LIN {X 0,Y 472.884,Z 110.578,A -85,B 0,C 180,E1 22845.551,E2 22845.551} C_VEL
LIN {X 0,Y 472.896,Z 110.565,A -85,B 0,C 180,E1 22842.019,E2 22842.019} C_VEL
LIN {X 0,Y 472.934,Z 110.57,A -85,B 0,C 180,E1 22838.468,E2 22838.468} C_VEL
LIN {X 0,Y 472.917,Z 110.572,A -85,B 0,C 180,E1 22834.851,E2 22834.851} C_VEL
LIN {X 0,Y 472.886,Z 110.562,A -85,B 0,C 180,E1 22831.317,E2 22831.317} C_VEL
LIN {X 0,Y 472.877,Z 110.572,A -85,B 0,C 180,E1 22827.752,E2 22827.752} C_VEL
LIN {X 0,Y 472.902,Z 110.576,A -85,B 0,C 180,E1 22824.279,E2 22824.279} C_VEL
LIN {X 0,Y 472.936,Z 110.577,A -85,B 0,C 180,E1 22820.636,E2 22820.636} C_VEL
LIN {X 0,Y 472.912,Z 110.58,A -85,B 0,C 180,E1 22817.014,E2 22817.014} C_VEL
LIN {X 0,Y 472.879,Z 110.58,A -85,B 0,C 180,E1 22813.511,E2 22813.511} C_VEL
LIN {X 0,Y 472.876,Z 110.577,A -85,B 0,C 180,E1 22809.867,E2 22809.867} C_VEL
LIN {X 0,Y 472.932,Z 110.708,A -85,B 0,C 180,E1 22806.545,E2 22806.545} C_VEL
LIN {X 0,Y 480.969,Z 132.457,A -85,B 0,C 180,E1 22803.528,E2 22803.528} C_VEL
LIN {X 0,Y 484.768,Z 144.05,A -85,B 0,C 180,E1 22802.036,E2 22802.036} C_VEL
LIN {X 0,Y 482.911,Z 174.424,A -85,B 0,C 180,E1 22799.238,E2 22799.238} C_VEL
LIN {X 0,Y 483.355,Z 176.82,A -85,B 0,C 180,E1 22799.166,E2 22799.166} C_VEL
LIN {X 0,Y 483.697,Z 184.5,A -85,B 0,C 180,E1 22799.017,E2 22799.017} C_VEL
LIN {X 0,Y 481.966,Z 196.735,A -85,B 0,C 180,E1 22798.947,E2 22798.947} C_VEL
LIN {X 0,Y 480.031,Z 209.081,A -85,B 0,C 180,E1 22798.891,E2 22798.891} C_VEL
LIN {X 0,Y 479.862,Z 212.462,A -85,B 0,C 180,E1 22798.849,E2 22798.849} C_VEL
LIN {X 0,Y 477.924,Z 389.612,A -85,B 0,C 180,E1 22796.211,E2 22796.211} C_VEL
LIN {X 0,Y 477.296,Z 408.622,A -85,B 0,C 180,E1 22795.702,E2 22795.702} C_VEL
LIN {X 0,Y 476.379,Z 426.597,A -85,B 0,C 180,E1 22794.998,E2 22794.998} C_VEL
LIN {X 0,Y 475.201,Z 443.939,A -85,B 0,C 180,E1 22794.09,E2 22794.09} C_VEL
LIN {X 0,Y 473.813,Z 460.62,A -85,B 0,C 180,E1 22792.978,E2 22792.978} C_VEL
LIN {X 0,Y 472.296,Z 476.507,A -85,B 0,C 180,E1 22791.662,E2 22791.662} C_VEL
LIN {X 0,Y 470.707,Z 491.623,A -85,B 0,C 180,E1 22790.127,E2 22790.127} C_VEL
LIN {X 0,Y 469.264,Z 504.803,A -85,B 0,C 180,E1 22788.509,E2 22788.509} C_VEL
LIN {X 0,Y 467.857,Z 517.403,A -85,B 0,C 180,E1 22786.64,E2 22786.64} C_VEL
LIN {X 0,Y 466.665,Z 528.464,A -85,B 0,C 180,E1 22784.644,E2 22784.644} C_VEL
LIN {X 0,Y 465.712,Z 538.034,A -85,B 0,C 180,E1 22782.523,E2 22782.523} C_VEL
LIN {X 0,Y 465.004,Z 546.099,A -85,B 0,C 180,E1 22780.28,E2 22780.28} C_VEL
LIN {X 0,Y 464.565,Z 552.332,A -85,B 0,C 180,E1 22778.041,E2 22778.041} C_VEL
LIN {X 0,Y 464.288,Z 557.107,A -85,B 0,C 180,E1 22775.684,E2 22775.684} C_VEL
LIN {X 0,Y 464.151,Z 560.185,A -85,B 0,C 180,E1 22773.334,E2 22773.334} C_VEL
LIN {X 0,Y 464.105,Z 561.659,A -85,B 0,C 180,E1 22770.987,E2 22770.987} C_VEL
LIN {X 0,Y 464.108,Z 561.574,A -85,B 0,C 180,E1 22768.641,E2 22768.641} C_VEL
LIN {X 0,Y 464.165,Z 559.923,A -85,B 0,C 180,E1 22766.294,E2 22766.294} C_VEL
LIN {X 0,Y 464.318,Z 556.648,A -85,B 0,C 180,E1 22763.942,E2 22763.942} C_VEL
LIN {X 0,Y 464.611,Z 551.647,A -85,B 0,C 180,E1 22761.584,E2 22761.584} C_VEL
LIN {X 0,Y 465.118,Z 544.77,A -85,B 0,C 180,E1 22759.22,E2 22759.22} C_VEL
LIN {X 0,Y 465.876,Z 536.323,A -85,B 0,C 180,E1 22756.976,E2 22756.976} C_VEL
LIN {X 0,Y 466.882,Z 526.333,A -85,B 0,C 180,E1 22754.854,E2 22754.854} C_VEL
LIN {X 0,Y 468.047,Z 515.598,A -85,B 0,C 180,E1 22752.982,E2 22752.982} C_VEL
LIN {X 0,Y 469.446,Z 503.079,A -85,B 0,C 180,E1 22751.175,E2 22751.175} C_VEL
LIN {X 0,Y 470.928,Z 489.575,A -85,B 0,C 180,E1 22749.557,E2 22749.557} C_VEL
LIN {X 0,Y 472.43,Z 475.214,A -85,B 0,C 180,E1 22748.13,E2 22748.13} C_VEL
LIN {X 0,Y 473.935,Z 459.24,A -85,B 0,C 180,E1 22746.829,E2 22746.829} C_VEL
LIN {X 0,Y 475.26,Z 443.306,A -85,B 0,C 180,E1 22745.779,E2 22745.779} C_VEL
LIN {X 0,Y 476.469,Z 425.323,A -85,B 0,C 180,E1 22744.852,E2 22744.852} C_VEL
LIN {X 0,Y 477.378,Z 406.697,A -85,B 0,C 180,E1 22744.143,E2 22744.143} C_VEL
LIN {X 0,Y 477.973,Z 387.762,A -85,B 0,C 180,E1 22743.661,E2 22743.661} C_VEL
LIN {X 0,Y 479.954,Z 196.45,A -85,B 0,C 180,E1 22740.803,E2 22740.803} C_VEL
LIN {X 0,Y 475.821,Z 173.604,A -85,B 0,C 180,E1 22740.096,E2 22740.096} C_VEL
LIN {X 0,Y 477.63,Z 146.449,A -85,B 0,C 180,E1 22737.526,E2 22737.526} C_VEL
LIN {X 0,Y 470.909,Z 127.236,A -85,B 0,C 180,E1 22734.937,E2 22734.937} C_VEL
LIN {X 0,Y 464.971,Z 111.558,A -85,B 0,C 180,E1 22732.631,E2 22732.631} C_VEL
LIN {X 0,Y 465.011,Z 111.552,A -85,B 0,C 180,E1 22729.181,E2 22729.181} C_VEL
LIN {X 0,Y 465.016,Z 111.564,A -85,B 0,C 180,E1 22725.496,E2 22725.496} C_VEL
LIN {X 0,Y 465.012,Z 111.562,A -85,B 0,C 180,E1 22721.744,E2 22721.744} C_VEL
LIN {X 0,Y 465.009,Z 111.563,A -85,B 0,C 180,E1 22718.096,E2 22718.096} C_VEL
LIN {X 0,Y 465.023,Z 111.688,A -85,B 0,C 180,E1 22715.488,E2 22715.488} C_VEL
LIN {X 0,Y 474.191,Z 138.149,A -85,B 0,C 180,E1 22712.496,E2 22712.496} C_VEL
LIN {X 0,Y 475.436,Z 142.809,A -85,B 0,C 180,E1 22712.003,E2 22712.003} C_VEL
LIN {X 0,Y 474.177,Z 181.693,A -85,B 0,C 180,E1 22708.738,E2 22708.738} C_VEL
LIN {X 0,Y 476.41,Z 196.928,A -85,B 0,C 180,E1 22708.313,E2 22708.313} C_VEL
LIN {X 0,Y 472.786,Z 392,A -85,B 0,C 180,E1 22704.905,E2 22704.905} C_VEL
LIN {X 0,Y 472.247,Z 411.513,A -85,B 0,C 180,E1 22704.331,E2 22704.331} C_VEL
LIN {X 0,Y 471.525,Z 429.876,A -85,B 0,C 180,E1 22703.56,E2 22703.56} C_VEL
LIN {X 0,Y 470.673,Z 447.161,A -85,B 0,C 180,E1 22702.613,E2 22702.613} C_VEL
LIN {X 0,Y 469.738,Z 463.701,A -85,B 0,C 180,E1 22701.476,E2 22701.476} C_VEL
LIN {X 0,Y 468.755,Z 479.425,A -85,B 0,C 180,E1 22700.15,E2 22700.15} C_VEL
LIN {X 0,Y 467.767,Z 494.215,A -85,B 0,C 180,E1 22698.637,E2 22698.637} C_VEL
LIN {X 0,Y 466.826,Z 507.992,A -85,B 0,C 180,E1 22696.935,E2 22696.935} C_VEL
LIN {X 0,Y 465.986,Z 520.624,A -85,B 0,C 180,E1 22695.048,E2 22695.048} C_VEL
LIN {X 0,Y 465.347,Z 531.015,A -85,B 0,C 180,E1 22693.165,E2 22693.165} C_VEL
LIN {X 0,Y 464.851,Z 540.065,A -85,B 0,C 180,E1 22691.162,E2 22691.162} C_VEL
LIN {X 0,Y 464.502,Z 547.713,A -85,B 0,C 180,E1 22689.041,E2 22689.041} C_VEL
LIN {X 0,Y 464.287,Z 553.881,A -85,B 0,C 180,E1 22686.803,E2 22686.803} C_VEL
LIN {X 0,Y 464.162,Z 558.237,A -85,B 0,C 180,E1 22684.572,E2 22684.572} C_VEL
LIN {X 0,Y 464.122,Z 560.897,A -85,B 0,C 180,E1 22682.346,E2 22682.346} C_VEL
LIN {X 0,Y 464.117,Z 561.965,A -85,B 0,C 180,E1 22680,E2 22680} C_VEL
LIN {X 0,Y 464.137,Z 561.22,A -85,B 0,C 180,E1 22677.654,E2 22677.654} C_VEL
LIN {X 0,Y 464.202,Z 558.846,A -85,B 0,C 180,E1 22675.429,E2 22675.429} C_VEL
LIN {X 0,Y 464.341,Z 554.769,A -85,B 0,C 180,E1 22673.199,E2 22673.199} C_VEL
LIN {X 0,Y 464.581,Z 548.874,A -85,B 0,C 180,E1 22670.961,E2 22670.961} C_VEL
LIN {X 0,Y 464.95,Z 541.471,A -85,B 0,C 180,E1 22668.841,E2 22668.841} C_VEL
LIN {X 0,Y 465.464,Z 532.625,A -85,B 0,C 180,E1 22666.839,E2 22666.839} C_VEL
LIN {X 0,Y 466.153,Z 521.688,A -85,B 0,C 180,E1 22664.844,E2 22664.844} C_VEL
LIN {X 0,Y 466.941,Z 509.853,A -85,B 0,C 180,E1 22663.069,E2 22663.069} C_VEL
LIN {X 0,Y 467.832,Z 496.357,A -85,B 0,C 180,E1 22661.398,E2 22661.398} C_VEL
LIN {X 0,Y 468.744,Z 481.822,A -85,B 0,C 180,E1 22659.915,E2 22659.915} C_VEL
LIN {X 0,Y 469.664,Z 466.017,A -85,B 0,C 180,E1 22658.586,E2 22658.586} C_VEL
LIN {X 0,Y 470.528,Z 449.162,A -85,B 0,C 180,E1 22657.441,E2 22657.441} C_VEL
LIN {X 0,Y 471.258,Z 431.359,A -85,B 0,C 180,E1 22656.492,E2 22656.492} C_VEL
LIN {X 0,Y 471.838,Z 412.338,A -85,B 0,C 180,E1 22655.73,E2 22655.73} C_VEL
LIN {X 0,Y 472.248,Z 392.418,A -85,B 0,C 180,E1 22655.181,E2 22655.181} C_VEL
LIN {X 0,Y 474.476,Z 285.661,A -85,B 0,C 180,E1 22653.199,E2 22653.199} C_VEL
LIN {X 0,Y 477.349,Z 195.104,A -85,B 0,C 180,E1 22651.339,E2 22651.339} C_VEL
LIN {X 0,Y 476.497,Z 189.323,A -85,B 0,C 180,E1 22651.106,E2 22651.106} C_VEL
LIN {X 0,Y 477.357,Z 150.37,A -85,B 0,C 180,E1 22648,E2 22648} C_VEL
LIN {X 0,Y 477.285,Z 141.627,A -85,B 0,C 180,E1 22647.284,E2 22647.284} C_VEL
LIN {X 0,Y 473.092,Z 129.321,A -85,B 0,C 180,E1 22645.835,E2 22645.835} C_VEL
LIN {X 0,Y 468.871,Z 119.813,A -85,B 0,C 180,E1 22644.547,E2 22644.547} C_VEL
LIN {X 0,Y 466.651,Z 115.532,A -85,B 0,C 180,E1 22643.898,E2 22643.898} C_VEL
LIN {X 0,Y 465.172,Z 112.443,A -85,B 0,C 180,E1 22643.429,E2 22643.429} C_VEL
LIN {X 0,Y 465.004,Z 111.566,A -85,B 0,C 180,E1 22643.291,E2 22643.291} C_VEL
LIN {X 0,Y 465.017,Z 111.564,A -85,B 0,C 180,E1 22639.567,E2 22639.567} C_VEL
LIN {X 0,Y 464.995,Z 111.566,A -85,B 0,C 180,E1 22635.839,E2 22635.839} C_VEL
LIN {X 0,Y 464.957,Z 111.57,A -85,B 0,C 180,E1 22632.29,E2 22632.29} C_VEL
LIN {X 0,Y 464.98,Z 111.74,A -85,B 0,C 180,E1 22631.259,E2 22631.259} C_VEL
LIN {X 0,Y 466.342,Z 115.196,A -85,B 0,C 180,E1 22630.813,E2 22630.813} C_VEL
LIN {X 0,Y 474.889,Z 135.664,A -85,B 0,C 180,E1 22628.244,E2 22628.244} C_VEL
LIN {X 0,Y 480.318,Z 150.221,A -85,B 0,C 180,E1 22626.579,E2 22626.579} C_VEL
LIN {X 0,Y 479.458,Z 164.644,A -85,B 0,C 180,E1 22625.503,E2 22625.503} C_VEL
LIN {X 0,Y 482.328,Z 186.5,A -85,B 0,C 180,E1 22624.889,E2 22624.889} C_VEL
LIN {X 0,Y 477.886,Z 419.576,A -85,B 0,C 180,E1 22620.981,E2 22620.981} C_VEL
LIN {X 0,Y 477.06,Z 440.311,A -85,B 0,C 180,E1 22620.457,E2 22620.457} C_VEL
LIN {X 0,Y 475.912,Z 461.474,A -85,B 0,C 180,E1 22619.697,E2 22619.697} C_VEL
LIN {X 0,Y 474.61,Z 482.255,A -85,B 0,C 180,E1 22618.707,E2 22618.707} C_VEL
LIN {X 0,Y 473.221,Z 501.389,A -85,B 0,C 180,E1 22617.564,E2 22617.564} C_VEL
LIN {X 0,Y 471.864,Z 519.025,A -85,B 0,C 180,E1 22616.287,E2 22616.287} C_VEL
LIN {X 0,Y 470.379,Z 537.148,A -85,B 0,C 180,E1 22614.713,E2 22614.713} C_VEL
LIN {X 0,Y 468.909,Z 554.52,A -85,B 0,C 180,E1 22612.905,E2 22612.905} C_VEL
LIN {X 0,Y 467.617,Z 569.978,A -85,B 0,C 180,E1 22610.987,E2 22610.987} C_VEL
LIN {X 0,Y 466.549,Z 583.421,A -85,B 0,C 180,E1 22609.012,E2 22609.012} C_VEL
LIN {X 0,Y 465.633,Z 595.835,A -85,B 0,C 180,E1 22606.852,E2 22606.852} C_VEL
LIN {X 0,Y 464.941,Z 606.773,A -85,B 0,C 180,E1 22604.573,E2 22604.573} C_VEL
LIN {X 0,Y 464.464,Z 615.766,A -85,B 0,C 180,E1 22602.306,E2 22602.306} C_VEL
LIN {X 0,Y 464.166,Z 623.312,A -85,B 0,C 180,E1 22599.924,E2 22599.924} C_VEL
LIN {X 0,Y 464,Z 629.057,A -85,B 0,C 180,E1 22597.554,E2 22597.554} C_VEL
LIN {X 0,Y 463.931,Z 633.365,A -85,B 0,C 180,E1 22595.07,E2 22595.07} C_VEL
LIN {X 0,Y 463.909,Z 635.899,A -85,B 0,C 180,E1 22592.719,E2 22592.719} C_VEL
LIN {X 0,Y 463.906,Z 636.873,A -85,B 0,C 180,E1 22590.248,E2 22590.248} C_VEL
LIN {X 0,Y 463.907,Z 636.257,A -85,B 0,C 180,E1 22587.901,E2 22587.901} C_VEL
LIN {X 0,Y 463.918,Z 634.033,A -85,B 0,C 180,E1 22585.427,E2 22585.427} C_VEL
LIN {X 0,Y 463.987,Z 630.124,A -85,B 0,C 180,E1 22582.945,E2 22582.945} C_VEL
LIN {X 0,Y 464.139,Z 624.343,A -85,B 0,C 180,E1 22580.453,E2 22580.453} C_VEL
LIN {X 0,Y 464.41,Z 617.058,A -85,B 0,C 180,E1 22578.073,E2 22578.073} C_VEL
LIN {X 0,Y 464.876,Z 607.875,A -85,B 0,C 180,E1 22575.681,E2 22575.681} C_VEL
LIN {X 0,Y 465.546,Z 597.191,A -85,B 0,C 180,E1 22573.403,E2 22573.403} C_VEL
LIN {X 0,Y 466.43,Z 585.055,A -85,B 0,C 180,E1 22571.245,E2 22571.245} C_VEL
LIN {X 0,Y 467.536,Z 571.073,A -85,B 0,C 180,E1 22569.156,E2 22569.156} C_VEL
LIN {X 0,Y 468.863,Z 555.12,A -85,B 0,C 180,E1 22567.164,E2 22567.164} C_VEL
LIN {X 0,Y 470.301,Z 538.046,A -85,B 0,C 180,E1 22565.375,E2 22565.375} C_VEL
LIN {X 0,Y 471.763,Z 520.178,A -85,B 0,C 180,E1 22563.807,E2 22563.807} C_VEL
LIN {X 0,Y 473.146,Z 502.356,A -85,B 0,C 180,E1 22562.502,E2 22562.502} C_VEL
LIN {X 0,Y 474.555,Z 483.031,A -85,B 0,C 180,E1 22561.335,E2 22561.335} C_VEL
LIN {X 0,Y 475.816,Z 463.201,A -85,B 0,C 180,E1 22560.375,E2 22560.375} C_VEL
LIN {X 0,Y 476.949,Z 442.8,A -85,B 0,C 180,E1 22559.617,E2 22559.617} C_VEL
LIN {X 0,Y 477.827,Z 421.76,A -85,B 0,C 180,E1 22559.06,E2 22559.06} C_VEL
LIN {X 0,Y 482.199,Z 192.981,A -85,B 0,C 180,E1 22555.217,E2 22555.217} C_VEL
LIN {X 0,Y 482.153,Z 183.797,A -85,B 0,C 180,E1 22555.048,E2 22555.048} C_VEL
LIN {X 0,Y 479.375,Z 163.766,A -85,B 0,C 180,E1 22554.465,E2 22554.465} C_VEL
LIN {X 0,Y 480.247,Z 149.701,A -85,B 0,C 180,E1 22553.379,E2 22553.379} C_VEL
LIN {X 0,Y 472.083,Z 128.682,A -85,B 0,C 180,E1 22550.917,E2 22550.917} C_VEL
LIN {X 0,Y 465.849,Z 114.357,A -85,B 0,C 180,E1 22549.069,E2 22549.069} C_VEL
LIN {X 0,Y 464.971,Z 111.558,A -85,B 0,C 180,E1 22548.689,E2 22548.689} C_VEL
LIN {X 0,Y 464.959,Z 111.567,A -85,B 0,C 180,E1 22545.145,E2 22545.145} C_VEL
LIN {X 0,Y 464.967,Z 111.565,A -85,B 0,C 180,E1 22541.477,E2 22541.477} C_VEL
LIN {X 0,Y 464.989,Z 111.522,A -85,B 0,C 180,E1 22537.895,E2 22537.895} C_VEL
LIN {X 0,Y 465.005,Z 111.562,A -85,B 0,C 180,E1 22534.288,E2 22534.288} C_VEL
LIN {X 0,Y 464.98,Z 111.565,A -85,B 0,C 180,E1 22530.639,E2 22530.639} C_VEL
LIN {X 0,Y 464.956,Z 111.564,A -85,B 0,C 180,E1 22527.094,E2 22527.094} C_VEL
LIN {X 0,Y 464.955,Z 111.557,A -85,B 0,C 180,E1 22523.442,E2 22523.442} C_VEL
LIN {X 0,Y 464.986,Z 111.555,A -85,B 0,C 180,E1 22519.992,E2 22519.992} C_VEL
LIN {X 0,Y 465.005,Z 111.562,A -85,B 0,C 180,E1 22516.36,E2 22516.36} C_VEL
LIN {X 0,Y 464.97,Z 111.547,A -85,B 0,C 180,E1 22512.796,E2 22512.796} C_VEL
LIN {X 0,Y 464.951,Z 111.564,A -85,B 0,C 180,E1 22509.234,E2 22509.234} C_VEL
LIN {X 0,Y 464.95,Z 111.563,A -85,B 0,C 180,E1 22505.553,E2 22505.553} C_VEL
LIN {X 0,Y 464.967,Z 111.552,A -85,B 0,C 180,E1 22501.971,E2 22501.971} C_VEL
LIN {X 0,Y 465.001,Z 111.562,A -85,B 0,C 180,E1 22498.398,E2 22498.398} C_VEL
LIN {X 0,Y 464.985,Z 111.547,A -85,B 0,C 180,E1 22494.694,E2 22494.694} C_VEL
LIN {X 0,Y 464.952,Z 111.566,A -85,B 0,C 180,E1 22491.217,E2 22491.217} C_VEL
LIN {X 0,Y 464.946,Z 111.557,A -85,B 0,C 180,E1 22487.581,E2 22487.581} C_VEL
LIN {X 0,Y 464.956,Z 111.56,A -85,B 0,C 180,E1 22483.993,E2 22483.993} C_VEL
LIN {X 0,Y 464.988,Z 111.563,A -85,B 0,C 180,E1 22480.4,E2 22480.4} C_VEL
LIN {X 0,Y 464.981,Z 111.549,A -85,B 0,C 180,E1 22476.827,E2 22476.827} C_VEL
LIN {X 0,Y 464.949,Z 111.565,A -85,B 0,C 180,E1 22473.291,E2 22473.291} C_VEL
LIN {X 0,Y 464.941,Z 111.566,A -85,B 0,C 180,E1 22469.787,E2 22469.787} C_VEL
LIN {X 0,Y 464.966,Z 111.558,A -85,B 0,C 180,E1 22466.303,E2 22466.303} C_VEL
LIN {X 0,Y 464.989,Z 111.555,A -85,B 0,C 180,E1 22462.671,E2 22462.671} C_VEL
LIN {X 0,Y 464.957,Z 111.561,A -85,B 0,C 180,E1 22459.176,E2 22459.176} C_VEL
LIN {X 0,Y 464.937,Z 111.56,A -85,B 0,C 180,E1 22455.659,E2 22455.659} C_VEL
LIN {X 0,Y 464.94,Z 111.571,A -85,B 0,C 180,E1 22451.92,E2 22451.92} C_VEL
LIN {X 0,Y 464.964,Z 111.566,A -85,B 0,C 180,E1 22448.422,E2 22448.422} C_VEL
LIN {X 0,Y 464.964,Z 111.582,A -85,B 0,C 180,E1 22447.234,E2 22447.234} C_VEL
LIN {X 0,Y 473.344,Z 133.939,A -85,B 0,C 180,E1 22444.039,E2 22444.039} C_VEL
LIN {X 0,Y 477.642,Z 146.882,A -85,B 0,C 180,E1 22442.332,E2 22442.332} C_VEL
LIN {X 0,Y 475.862,Z 174.32,A -85,B 0,C 180,E1 22439.775,E2 22439.775} C_VEL
LIN {X 0,Y 480.041,Z 198.192,A -85,B 0,C 180,E1 22439.066,E2 22439.066} C_VEL
LIN {X 0,Y 479.862,Z 212.462,A -85,B 0,C 180,E1 22438.849,E2 22438.849} C_VEL
LIN {X 0,Y 478.922,Z 220.158,A -85,B 0,C 180,E1 22438.796,E2 22438.796} C_VEL
LIN {X 0,Y 473.357,Z 240.654,A -85,B 0,C 180,E1 22438.882,E2 22438.882} C_VEL
LIN {X 0,Y 472.632,Z 247.261,A -85,B 0,C 180,E1 22438.83,E2 22438.83} C_VEL
LIN {X 0,Y 470.941,Z 389.942,A -85,B 0,C 180,E1 22436.681,E2 22436.681} C_VEL
LIN {X 0,Y 470.272,Z 408.97,A -85,B 0,C 180,E1 22436.166,E2 22436.166} C_VEL
LIN {X 0,Y 469.353,Z 426.237,A -85,B 0,C 180,E1 22435.487,E2 22435.487} C_VEL
LIN {X 0,Y 468.072,Z 444.088,A -85,B 0,C 180,E1 22434.548,E2 22434.548} C_VEL
LIN {X 0,Y 466.596,Z 460.843,A -85,B 0,C 180,E1 22433.421,E2 22433.421} C_VEL
LIN {X 0,Y 464.942,Z 477.199,A -85,B 0,C 180,E1 22432.048,E2 22432.048} C_VEL
LIN {X 0,Y 463.255,Z 492.276,A -85,B 0,C 180,E1 22430.492,E2 22430.492} C_VEL
LIN {X 0,Y 461.691,Z 505.63,A -85,B 0,C 180,E1 22428.824,E2 22428.824} C_VEL
LIN {X 0,Y 460.19,Z 518.191,A -85,B 0,C 180,E1 22426.925,E2 22426.925} C_VEL
LIN {X 0,Y 458.914,Z 529.22,A -85,B 0,C 180,E1 22424.897,E2 22424.897} C_VEL
LIN {X 0,Y 457.889,Z 538.763,A -85,B 0,C 180,E1 22422.74,E2 22422.74} C_VEL
LIN {X 0,Y 457.122,Z 546.805,A -85,B 0,C 180,E1 22420.459,E2 22420.459} C_VEL
LIN {X 0,Y 456.64,Z 553.016,A -85,B 0,C 180,E1 22418.181,E2 22418.181} C_VEL
LIN {X 0,Y 456.336,Z 557.773,A -85,B 0,C 180,E1 22415.784,E2 22415.784} C_VEL
LIN {X 0,Y 456.183,Z 560.838,A -85,B 0,C 180,E1 22413.392,E2 22413.392} C_VEL
LIN {X 0,Y 456.132,Z 562.305,A -85,B 0,C 180,E1 22411.004,E2 22411.004} C_VEL
LIN {X 0,Y 456.135,Z 562.22,A -85,B 0,C 180,E1 22408.618,E2 22408.618} C_VEL
LIN {X 0,Y 456.2,Z 560.578,A -85,B 0,C 180,E1 22406.229,E2 22406.229} C_VEL
LIN {X 0,Y 456.369,Z 557.318,A -85,B 0,C 180,E1 22403.836,E2 22403.836} C_VEL
LIN {X 0,Y 456.692,Z 552.337,A -85,B 0,C 180,E1 22401.437,E2 22401.437} C_VEL
LIN {X 0,Y 457.247,Z 545.482,A -85,B 0,C 180,E1 22399.032,E2 22399.032} C_VEL
LIN {X 0,Y 458.068,Z 537.062,A -85,B 0,C 180,E1 22396.75,E2 22396.75} C_VEL
LIN {X 0,Y 459.081,Z 527.764,A -85,B 0,C 180,E1 22394.719,E2 22394.719} C_VEL
LIN {X 0,Y 460.398,Z 516.398,A -85,B 0,C 180,E1 22392.69,E2 22392.69} C_VEL
LIN {X 0,Y 461.89,Z 503.92,A -85,B 0,C 180,E1 22390.855,E2 22390.855} C_VEL
LIN {X 0,Y 463.467,Z 490.469,A -85,B 0,C 180,E1 22389.213,E2 22389.213} C_VEL
LIN {X 0,Y 465.132,Z 475.466,A -85,B 0,C 180,E1 22387.702,E2 22387.702} C_VEL
LIN {X 0,Y 466.73,Z 459.427,A -85,B 0,C 180,E1 22386.383,E2 22386.383} C_VEL
LIN {X 0,Y 468.135,Z 443.413,A -85,B 0,C 180,E1 22385.319,E2 22385.319} C_VEL
LIN {X 0,Y 469.417,Z 425.305,A -85,B 0,C 180,E1 22384.38,E2 22384.38} C_VEL
LIN {X 0,Y 470.363,Z 407.017,A -85,B 0,C 180,E1 22383.678,E2 22383.678} C_VEL
LIN {X 0,Y 470.994,Z 388.14,A -85,B 0,C 180,E1 22383.191,E2 22383.191} C_VEL
LIN {X 0,Y 473.154,Z 197.742,A -85,B 0,C 180,E1 22380.307,E2 22380.307} C_VEL
LIN {X 0,Y 468.812,Z 173.404,A -85,B 0,C 180,E1 22379.531,E2 22379.531} C_VEL
LIN {X 0,Y 470.557,Z 149.679,A -85,B 0,C 180,E1 22377.263,E2 22377.263} C_VEL
LIN {X 0,Y 463.949,Z 130.687,A -85,B 0,C 180,E1 22374.658,E2 22374.658} C_VEL
LIN {X 0,Y 458.059,Z 115.586,A -85,B 0,C 180,E1 22372.407,E2 22372.407} C_VEL
LIN {X 0,Y 457.042,Z 112.527,A -85,B 0,C 180,E1 22371.907,E2 22371.907} C_VEL
LIN {X 0,Y 457.05,Z 112.558,A -85,B 0,C 180,E1 22368.244,E2 22368.244} C_VEL
LIN {X 0,Y 457.054,Z 112.552,A -85,B 0,C 180,E1 22364.506,E2 22364.506} C_VEL
LIN {X 0,Y 457.063,Z 112.55,A -85,B 0,C 180,E1 22360.808,E2 22360.808} C_VEL
LIN {X 0,Y 457.072,Z 112.549,A -85,B 0,C 180,E1 22357.14,E2 22357.14} C_VEL
LIN {X 0,Y 457.076,Z 112.659,A -85,B 0,C 180,E1 22356.012,E2 22356.012} C_VEL
LIN {X 0,Y 466.199,Z 138.753,A -85,B 0,C 180,E1 22353.008,E2 22353.008} C_VEL
LIN {X 0,Y 468.16,Z 145.565,A -85,B 0,C 180,E1 22352.272,E2 22352.272} C_VEL
LIN {X 0,Y 466.936,Z 182.274,A -85,B 0,C 180,E1 22349.18,E2 22349.18} C_VEL
LIN {X 0,Y 469.217,Z 197.998,A -85,B 0,C 180,E1 22348.726,E2 22348.726} C_VEL
LIN {X 0,Y 465.316,Z 392.645,A -85,B 0,C 180,E1 22345.248,E2 22345.248} C_VEL
LIN {X 0,Y 464.745,Z 412.117,A -85,B 0,C 180,E1 22344.663,E2 22344.663} C_VEL
LIN {X 0,Y 463.956,Z 430.969,A -85,B 0,C 180,E1 22343.854,E2 22343.854} C_VEL
LIN {X 0,Y 463.044,Z 448.433,A -85,B 0,C 180,E1 22342.873,E2 22342.873} C_VEL
LIN {X 0,Y 462.02,Z 465.459,A -85,B 0,C 180,E1 22341.669,E2 22341.669} C_VEL
LIN {X 0,Y 460.933,Z 481.828,A -85,B 0,C 180,E1 22340.242,E2 22340.242} C_VEL
LIN {X 0,Y 459.909,Z 496.366,A -85,B 0,C 180,E1 22338.704,E2 22338.704} C_VEL
LIN {X 0,Y 458.94,Z 509.938,A -85,B 0,C 180,E1 22336.974,E2 22336.974} C_VEL
LIN {X 0,Y 458.123,Z 521.619,A -85,B 0,C 180,E1 22335.183,E2 22335.183} C_VEL
LIN {X 0,Y 457.449,Z 531.987,A -85,B 0,C 180,E1 22333.268,E2 22333.268} C_VEL
LIN {X 0,Y 456.924,Z 541.002,A -85,B 0,C 180,E1 22331.231,E2 22331.231} C_VEL
LIN {X 0,Y 456.553,Z 548.611,A -85,B 0,C 180,E1 22329.073,E2 22329.073} C_VEL
LIN {X 0,Y 456.324,Z 554.737,A -85,B 0,C 180,E1 22326.795,E2 22326.795} C_VEL
LIN {X 0,Y 456.193,Z 559.047,A -85,B 0,C 180,E1 22324.526,E2 22324.526} C_VEL
LIN {X 0,Y 456.147,Z 561.743,A -85,B 0,C 180,E1 22322.136,E2 22322.136} C_VEL
LIN {X 0,Y 456.147,Z 562.631,A -85,B 0,C 180,E1 22319.875,E2 22319.875} C_VEL
LIN {X 0,Y 456.169,Z 561.903,A -85,B 0,C 180,E1 22317.613,E2 22317.613} C_VEL
LIN {X 0,Y 456.245,Z 559.537,A -85,B 0,C 180,E1 22315.349,E2 22315.349} C_VEL
LIN {X 0,Y 456.401,Z 555.462,A -85,B 0,C 180,E1 22313.08,E2 22313.08} C_VEL
LIN {X 0,Y 456.652,Z 549.935,A -85,B 0,C 180,E1 22310.928,E2 22310.928} C_VEL
LIN {X 0,Y 457.047,Z 542.607,A -85,B 0,C 180,E1 22308.773,E2 22308.773} C_VEL
LIN {X 0,Y 457.6,Z 533.846,A -85,B 0,C 180,E1 22306.737,E2 22306.737} C_VEL
LIN {X 0,Y 458.294,Z 523.711,A -85,B 0,C 180,E1 22304.823,E2 22304.823} C_VEL
LIN {X 0,Y 459.109,Z 512.192,A -85,B 0,C 180,E1 22303.033,E2 22303.033} C_VEL
LIN {X 0,Y 460.06,Z 498.707,A -85,B 0,C 180,E1 22301.303,E2 22301.303} C_VEL
LIN {X 0,Y 461.053,Z 484.195,A -85,B 0,C 180,E1 22299.764,E2 22299.764} C_VEL
LIN {X 0,Y 462.02,Z 468.677,A -85,B 0,C 180,E1 22298.414,E2 22298.414} C_VEL
LIN {X 0,Y 462.98,Z 451.328,A -85,B 0,C 180,E1 22297.192,E2 22297.192} C_VEL
LIN {X 0,Y 463.8,Z 433.347,A -85,B 0,C 180,E1 22296.192,E2 22296.192} C_VEL
LIN {X 0,Y 464.438,Z 414.471,A -85,B 0,C 180,E1 22295.407,E2 22295.407} C_VEL
LIN {X 0,Y 464.877,Z 395.153,A -85,B 0,C 180,E1 22294.846,E2 22294.846} C_VEL
LIN {X 0,Y 467.441,Z 286.91,A -85,B 0,C 180,E1 22292.75,E2 22292.75} C_VEL
LIN {X 0,Y 470.714,Z 196.563,A -85,B 0,C 180,E1 22290.821,E2 22290.821} C_VEL
LIN {X 0,Y 469.842,Z 190.427,A -85,B 0,C 180,E1 22290.555,E2 22290.555} C_VEL
LIN {X 0,Y 470.904,Z 150.854,A -85,B 0,C 180,E1 22287.363,E2 22287.363} C_VEL
LIN {X 0,Y 470.942,Z 145.552,A -85,B 0,C 180,E1 22286.932,E2 22286.932} C_VEL
LIN {X 0,Y 467.085,Z 133.878,A -85,B 0,C 180,E1 22285.503,E2 22285.503} C_VEL
LIN {X 0,Y 463.004,Z 124.623,A -85,B 0,C 180,E1 22284.181,E2 22284.181} C_VEL
LIN {X 0,Y 460.946,Z 120.589,A -85,B 0,C 180,E1 22283.534,E2 22283.534} C_VEL
LIN {X 0,Y 459.44,Z 117.337,A -85,B 0,C 180,E1 22283.006,E2 22283.006} C_VEL
LIN {X 0,Y 457.514,Z 114.475,A -85,B 0,C 180,E1 22282.43,E2 22282.43} C_VEL
LIN {X 0,Y 457.037,Z 112.557,A -85,B 0,C 180,E1 22282.164,E2 22282.164} C_VEL
LIN {X 0,Y 457.019,Z 112.558,A -85,B 0,C 180,E1 22278.627,E2 22278.627} C_VEL
LIN {X 0,Y 457.017,Z 112.559,A -85,B 0,C 180,E1 22274.964,E2 22274.964} C_VEL
LIN {X 0,Y 457.059,Z 112.687,A -85,B 0,C 180,E1 22271.987,E2 22271.987} C_VEL
LIN {X 0,Y 466.971,Z 136.342,A -85,B 0,C 180,E1 22268.894,E2 22268.894} C_VEL
LIN {X 0,Y 473.279,Z 153.219,A -85,B 0,C 180,E1 22266.907,E2 22266.907} C_VEL
LIN {X 0,Y 472.536,Z 164.63,A -85,B 0,C 180,E1 22266.042,E2 22266.042} C_VEL
LIN {X 0,Y 475.524,Z 187.757,A -85,B 0,C 180,E1 22265.38,E2 22265.38} C_VEL
LIN {X 0,Y 470.836,Z 417.194,A -85,B 0,C 180,E1 22261.47,E2 22261.47} C_VEL
LIN {X 0,Y 469.928,Z 438.77,A -85,B 0,C 180,E1 22260.931,E2 22260.931} C_VEL
LIN {X 0,Y 468.703,Z 460.13,A -85,B 0,C 180,E1 22260.158,E2 22260.158} C_VEL
LIN {X 0,Y 467.337,Z 480.17,A -85,B 0,C 180,E1 22259.197,E2 22259.197} C_VEL
LIN {X 0,Y 465.85,Z 499.461,A -85,B 0,C 180,E1 22258.038,E2 22258.038} C_VEL
LIN {X 0,Y 464.302,Z 518.311,A -85,B 0,C 180,E1 22256.66,E2 22256.66} C_VEL
LIN {X 0,Y 462.72,Z 536.497,A -85,B 0,C 180,E1 22255.058,E2 22255.058} C_VEL
LIN {X 0,Y 461.179,Z 553.712,A -85,B 0,C 180,E1 22253.241,E2 22253.241} C_VEL
LIN {X 0,Y 459.814,Z 569.203,A -85,B 0,C 180,E1 22251.294,E2 22251.294} C_VEL
LIN {X 0,Y 458.69,Z 582.684,A -85,B 0,C 180,E1 22249.291,E2 22249.291} C_VEL
LIN {X 0,Y 457.745,Z 594.893,A -85,B 0,C 180,E1 22247.151,E2 22247.151} C_VEL
LIN {X 0,Y 457.042,Z 605.379,A -85,B 0,C 180,E1 22244.961,E2 22244.961} C_VEL
LIN {X 0,Y 456.523,Z 614.532,A -85,B 0,C 180,E1 22242.652,E2 22242.652} C_VEL
LIN {X 0,Y 456.197,Z 622.19,A -85,B 0,C 180,E1 22240.227,E2 22240.227} C_VEL
LIN {X 0,Y 456.029,Z 628.081,A -85,B 0,C 180,E1 22237.814,E2 22237.814} C_VEL
LIN {X 0,Y 455.952,Z 632.382,A -85,B 0,C 180,E1 22235.392,E2 22235.392} C_VEL
LIN {X 0,Y 455.936,Z 635.165,A -85,B 0,C 180,E1 22232.892,E2 22232.892} C_VEL
LIN {X 0,Y 455.929,Z 636.204,A -85,B 0,C 180,E1 22230.378,E2 22230.378} C_VEL
LIN {X 0,Y 455.93,Z 635.608,A -85,B 0,C 180,E1 22227.864,E2 22227.864} C_VEL
LIN {X 0,Y 455.94,Z 633.365,A -85,B 0,C 180,E1 22225.347,E2 22225.347} C_VEL
LIN {X 0,Y 456,Z 629.662,A -85,B 0,C 180,E1 22222.948,E2 22222.948} C_VEL
LIN {X 0,Y 456.138,Z 624.249,A -85,B 0,C 180,E1 22220.538,E2 22220.538} C_VEL
LIN {X 0,Y 456.404,Z 617.122,A -85,B 0,C 180,E1 22218.117,E2 22218.117} C_VEL
LIN {X 0,Y 456.872,Z 608.101,A -85,B 0,C 180,E1 22215.683,E2 22215.683} C_VEL
LIN {X 0,Y 457.558,Z 597.588,A -85,B 0,C 180,E1 22213.367,E2 22213.367} C_VEL
LIN {X 0,Y 458.467,Z 585.567,A -85,B 0,C 180,E1 22211.17,E2 22211.17} C_VEL
LIN {X 0,Y 459.575,Z 572.023,A -85,B 0,C 180,E1 22209.097,E2 22209.097} C_VEL
LIN {X 0,Y 460.888,Z 556.994,A -85,B 0,C 180,E1 22207.151,E2 22207.151} C_VEL
LIN {X 0,Y 462.359,Z 540.384,A -85,B 0,C 180,E1 22205.333,E2 22205.333} C_VEL
LIN {X 0,Y 463.892,Z 522.847,A -85,B 0,C 180,E1 22203.719,E2 22203.719} C_VEL
LIN {X 0,Y 465.466,Z 504.092,A -85,B 0,C 180,E1 22202.28,E2 22202.28} C_VEL
LIN {X 0,Y 466.993,Z 484.85,A -85,B 0,C 180,E1 22201.062,E2 22201.062} C_VEL
LIN {X 0,Y 468.359,Z 465.741,A -85,B 0,C 180,E1 22200.081,E2 22200.081} C_VEL
LIN {X 0,Y 469.677,Z 444.145,A -85,B 0,C 180,E1 22199.234,E2 22199.234} C_VEL
LIN {X 0,Y 470.673,Z 422.422,A -85,B 0,C 180,E1 22198.634,E2 22198.634} C_VEL
LIN {X 0,Y 474.353,Z 243.277,A -85,B 0,C 180,E1 22195.558,E2 22195.558} C_VEL
LIN {X 0,Y 475.367,Z 185.098,A -85,B 0,C 180,E1 22194.559,E2 22194.559} C_VEL
LIN {X 0,Y 472.499,Z 163.486,A -85,B 0,C 180,E1 22193.899,E2 22193.899} C_VEL
LIN {X 0,Y 473.09,Z 152.487,A -85,B 0,C 180,E1 22193.024,E2 22193.024} C_VEL
LIN {X 0,Y 465.446,Z 132.704,A -85,B 0,C 180,E1 22190.655,E2 22190.655} C_VEL
LIN {X 0,Y 458.279,Z 115.916,A -85,B 0,C 180,E1 22188.447,E2 22188.447} C_VEL
LIN {X 0,Y 457.065,Z 112.544,A -85,B 0,C 180,E1 22187.981,E2 22187.981} C_VEL
LIN {X 0,Y 457.066,Z 112.551,A -85,B 0,C 180,E1 22184.253,E2 22184.253} C_VEL
LIN {X 0,Y 457.039,Z 112.54,A -85,B 0,C 180,E1 22180.614,E2 22180.614} C_VEL
LIN {X 0,Y 457.019,Z 112.529,A -85,B 0,C 180,E1 22176.987,E2 22176.987} C_VEL
LIN {X 0,Y 457.018,Z 112.544,A -85,B 0,C 180,E1 22173.307,E2 22173.307} C_VEL
LIN {X 0,Y 457.034,Z 112.547,A -85,B 0,C 180,E1 22169.715,E2 22169.715} C_VEL
LIN {X 0,Y 457.066,Z 112.554,A -85,B 0,C 180,E1 22166.224,E2 22166.224} C_VEL
LIN {X 0,Y 457.056,Z 112.545,A -85,B 0,C 180,E1 22162.509,E2 22162.509} C_VEL
LIN {X 0,Y 457.023,Z 112.539,A -85,B 0,C 180,E1 22158.892,E2 22158.892} C_VEL
LIN {X 0,Y 457.013,Z 112.554,A -85,B 0,C 180,E1 22155.246,E2 22155.246} C_VEL
LIN {X 0,Y 457.013,Z 112.553,A -85,B 0,C 180,E1 22151.484,E2 22151.484} C_VEL
LIN {X 0,Y 457.029,Z 112.537,A -85,B 0,C 180,E1 22147.922,E2 22147.922} C_VEL
LIN {X 0,Y 457.06,Z 112.553,A -85,B 0,C 180,E1 22144.391,E2 22144.391} C_VEL
LIN {X 0,Y 457.051,Z 112.533,A -85,B 0,C 180,E1 22140.626,E2 22140.626} C_VEL
LIN {X 0,Y 457.023,Z 112.555,A -85,B 0,C 180,E1 22136.99,E2 22136.99} C_VEL
LIN {X 0,Y 457.007,Z 112.547,A -85,B 0,C 180,E1 22133.344,E2 22133.344} C_VEL
LIN {X 0,Y 457.008,Z 112.547,A -85,B 0,C 180,E1 22129.665,E2 22129.665} C_VEL
LIN {X 0,Y 457.026,Z 112.556,A -85,B 0,C 180,E1 22126.075,E2 22126.075} C_VEL
LIN {X 0,Y 457.055,Z 112.535,A -85,B 0,C 180,E1 22122.512,E2 22122.512} C_VEL
LIN {X 0,Y 457.043,Z 112.555,A -85,B 0,C 180,E1 22118.84,E2 22118.84} C_VEL
LIN {X 0,Y 457.008,Z 112.549,A -85,B 0,C 180,E1 22115.299,E2 22115.299} C_VEL
LIN {X 0,Y 457.001,Z 112.538,A -85,B 0,C 180,E1 22111.655,E2 22111.655} C_VEL
LIN {X 0,Y 457.011,Z 112.549,A -85,B 0,C 180,E1 22108.031,E2 22108.031} C_VEL
LIN {X 0,Y 457.034,Z 112.554,A -85,B 0,C 180,E1 22104.413,E2 22104.413} C_VEL
LIN {X 0,Y 457.059,Z 112.555,A -85,B 0,C 180,E1 22100.75,E2 22100.75} C_VEL
LIN {X 0,Y 457.024,Z 112.558,A -85,B 0,C 180,E1 22097.125,E2 22097.125} C_VEL
LIN {X 0,Y 457.001,Z 112.559,A -85,B 0,C 180,E1 22093.564,E2 22093.564} C_VEL
LIN {X 0,Y 456.999,Z 112.554,A -85,B 0,C 180,E1 22089.83,E2 22089.83} C_VEL
LIN {X 0,Y 457.01,Z 112.625,A -85,B 0,C 180,E1 22087.935,E2 22087.935} C_VEL
LIN {X 0,Y 464.691,Z 132.895,A -85,B 0,C 180,E1 22084.936,E2 22084.936} C_VEL
LIN {X 0,Y 470.524,Z 149.806,A -85,B 0,C 180,E1 22082.629,E2 22082.629} C_VEL
LIN {X 0,Y 468.842,Z 174.176,A -85,B 0,C 180,E1 22080.33,E2 22080.33} C_VEL
LIN {X 0,Y 473.244,Z 199.517,A -85,B 0,C 180,E1 22079.559,E2 22079.559} C_VEL
LIN {X 0,Y 472.632,Z 247.261,A -85,B 0,C 180,E1 22078.83,E2 22078.83} C_VEL
LIN {X 0,Y 471.677,Z 254.959,A -85,B 0,C 180,E1 22078.779,E2 22078.779} C_VEL
LIN {X 0,Y 466.078,Z 275.444,A -85,B 0,C 180,E1 22078.873,E2 22078.873} C_VEL
LIN {X 0,Y 465.37,Z 282.05,A -85,B 0,C 180,E1 22078.821,E2 22078.821} C_VEL
LIN {X 0,Y 463.986,Z 390.269,A -85,B 0,C 180,E1 22077.164,E2 22077.164} C_VEL
LIN {X 0,Y 463.276,Z 409.314,A -85,B 0,C 180,E1 22076.643,E2 22076.643} C_VEL
LIN {X 0,Y 462.232,Z 427.572,A -85,B 0,C 180,E1 22075.908,E2 22075.908} C_VEL
LIN {X 0,Y 460.879,Z 445.216,A -85,B 0,C 180,E1 22074.957,E2 22074.957} C_VEL
LIN {X 0,Y 459.322,Z 461.848,A -85,B 0,C 180,E1 22073.815,E2 22073.815} C_VEL
LIN {X 0,Y 457.604,Z 477.887,A -85,B 0,C 180,E1 22072.444,E2 22072.444} C_VEL
LIN {X 0,Y 455.804,Z 493.03,A -85,B 0,C 180,E1 22070.855,E2 22070.855} C_VEL
LIN {X 0,Y 454.129,Z 506.438,A -85,B 0,C 180,E1 22069.15,E2 22069.15} C_VEL
LIN {X 0,Y 452.533,Z 518.961,A -85,B 0,C 180,E1 22067.221,E2 22067.221} C_VEL
LIN {X 0,Y 451.171,Z 529.963,A -85,B 0,C 180,E1 22065.158,E2 22065.158} C_VEL
LIN {X 0,Y 450.071,Z 539.48,A -85,B 0,C 180,E1 22062.965,E2 22062.965} C_VEL
LIN {X 0,Y 449.244,Z 547.501,A -85,B 0,C 180,E1 22060.644,E2 22060.644} C_VEL
LIN {X 0,Y 448.716,Z 553.693,A -85,B 0,C 180,E1 22058.327,E2 22058.327} C_VEL
LIN {X 0,Y 448.384,Z 558.435,A -85,B 0,C 180,E1 22055.887,E2 22055.887} C_VEL
LIN {X 0,Y 448.216,Z 561.489,A -85,B 0,C 180,E1 22053.452,E2 22053.452} C_VEL
LIN {X 0,Y 448.158,Z 562.95,A -85,B 0,C 180,E1 22051.022,E2 22051.022} C_VEL
LIN {X 0,Y 448.162,Z 562.867,A -85,B 0,C 180,E1 22048.593,E2 22048.593} C_VEL
LIN {X 0,Y 448.234,Z 561.231,A -85,B 0,C 180,E1 22046.162,E2 22046.162} C_VEL
LIN {X 0,Y 448.42,Z 557.983,A -85,B 0,C 180,E1 22043.727,E2 22043.727} C_VEL
LIN {X 0,Y 448.775,Z 553.019,A -85,B 0,C 180,E1 22041.285,E2 22041.285} C_VEL
LIN {X 0,Y 449.379,Z 546.185,A -85,B 0,C 180,E1 22038.838,E2 22038.838} C_VEL
LIN {X 0,Y 450.264,Z 537.786,A -85,B 0,C 180,E1 22036.516,E2 22036.516} C_VEL
LIN {X 0,Y 451.425,Z 527.851,A -85,B 0,C 180,E1 22034.322,E2 22034.322} C_VEL
LIN {X 0,Y 452.857,Z 516.374,A -85,B 0,C 180,E1 22032.26,E2 22032.26} C_VEL
LIN {X 0,Y 454.462,Z 503.771,A -85,B 0,C 180,E1 22030.395,E2 22030.395} C_VEL
LIN {X 0,Y 456.15,Z 490.169,A -85,B 0,C 180,E1 22028.729,E2 22028.729} C_VEL
LIN {X 0,Y 457.858,Z 475.697,A -85,B 0,C 180,E1 22027.261,E2 22027.261} C_VEL
LIN {X 0,Y 459.473,Z 460.467,A -85,B 0,C 180,E1 22025.987,E2 22025.987} C_VEL
LIN {X 0,Y 461.038,Z 443.487,A -85,B 0,C 180,E1 22024.844,E2 22024.844} C_VEL
LIN {X 0,Y 462.355,Z 425.994,A -85,B 0,C 180,E1 22023.925,E2 22023.925} C_VEL
LIN {X 0,Y 463.369,Z 407.504,A -85,B 0,C 180,E1 22023.204,E2 22023.204} C_VEL
LIN {X 0,Y 464.044,Z 388.461,A -85,B 0,C 180,E1 22022.706,E2 22022.706} C_VEL
LIN {X 0,Y 466.406,Z 199.094,A -85,B 0,C 180,E1 22019.8,E2 22019.8} C_VEL
LIN {X 0,Y 461.806,Z 173.56,A -85,B 0,C 180,E1 22018.982,E2 22018.982} C_VEL
LIN {X 0,Y 463.306,Z 152.261,A -85,B 0,C 180,E1 22016.906,E2 22016.906} C_VEL
LIN {X 0,Y 456.666,Z 133.133,A -85,B 0,C 180,E1 22014.225,E2 22014.225} C_VEL
LIN {X 0,Y 450.052,Z 116.376,A -85,B 0,C 180,E1 22011.651,E2 22011.651} C_VEL
LIN {X 0,Y 449.129,Z 113.503,A -85,B 0,C 180,E1 22011.186,E2 22011.186} C_VEL
LIN {X 0,Y 449.139,Z 113.537,A -85,B 0,C 180,E1 22007.465,E2 22007.465} C_VEL
LIN {X 0,Y 449.135,Z 113.529,A -85,B 0,C 180,E1 22003.654,E2 22003.654} C_VEL
LIN {X 0,Y 449.131,Z 113.541,A -85,B 0,C 180,E1 21999.878,E2 21999.878} C_VEL
LIN {X 0,Y 449.139,Z 113.581,A -85,B 0,C 180,E1 21996.552,E2 21996.552} C_VEL
LIN {X 0,Y 458.658,Z 140.674,A -85,B 0,C 180,E1 21993.391,E2 21993.391} C_VEL
LIN {X 0,Y 460.893,Z 148.33,A -85,B 0,C 180,E1 21992.549,E2 21992.549} C_VEL
LIN {X 0,Y 459.672,Z 182.682,A -85,B 0,C 180,E1 21989.634,E2 21989.634} C_VEL
LIN {X 0,Y 462.045,Z 199.118,A -85,B 0,C 180,E1 21989.15,E2 21989.15} C_VEL
LIN {X 0,Y 457.864,Z 393.251,A -85,B 0,C 180,E1 21985.602,E2 21985.602} C_VEL
LIN {X 0,Y 457.255,Z 412.812,A -85,B 0,C 180,E1 21985.002,E2 21985.002} C_VEL
LIN {X 0,Y 456.429,Z 431.555,A -85,B 0,C 180,E1 21984.183,E2 21984.183} C_VEL
LIN {X 0,Y 455.486,Z 448.714,A -85,B 0,C 180,E1 21983.206,E2 21983.206} C_VEL
LIN {X 0,Y 454.394,Z 465.996,A -85,B 0,C 180,E1 21981.967,E2 21981.967} C_VEL
LIN {X 0,Y 453.258,Z 482.228,A -85,B 0,C 180,E1 21980.533,E2 21980.533} C_VEL
LIN {X 0,Y 452.177,Z 496.818,A -85,B 0,C 180,E1 21978.969,E2 21978.969} C_VEL
LIN {X 0,Y 451.152,Z 510.41,A -85,B 0,C 180,E1 21977.214,E2 21977.214} C_VEL
LIN {X 0,Y 450.257,Z 522.553,A -85,B 0,C 180,E1 21975.323,E2 21975.323} C_VEL
LIN {X 0,Y 449.506,Z 533.537,A -85,B 0,C 180,E1 21973.245,E2 21973.245} C_VEL
LIN {X 0,Y 448.937,Z 542.895,A -85,B 0,C 180,E1 21971.043,E2 21971.043} C_VEL
LIN {X 0,Y 448.563,Z 550.242,A -85,B 0,C 180,E1 21968.848,E2 21968.848} C_VEL
LIN {X 0,Y 448.334,Z 556.098,A -85,B 0,C 180,E1 21966.531,E2 21966.531} C_VEL
LIN {X 0,Y 448.211,Z 560.162,A -85,B 0,C 180,E1 21964.222,E2 21964.222} C_VEL
LIN {X 0,Y 448.167,Z 562.536,A -85,B 0,C 180,E1 21961.918,E2 21961.918} C_VEL
LIN {X 0,Y 448.172,Z 563.279,A -85,B 0,C 180,E1 21959.617,E2 21959.617} C_VEL
LIN {X 0,Y 448.205,Z 562.391,A -85,B 0,C 180,E1 21957.315,E2 21957.315} C_VEL
LIN {X 0,Y 448.301,Z 559.848,A -85,B 0,C 180,E1 21955.01,E2 21955.01} C_VEL
LIN {X 0,Y 448.488,Z 555.571,A -85,B 0,C 180,E1 21952.7,E2 21952.7} C_VEL
LIN {X 0,Y 448.803,Z 549.446,A -85,B 0,C 180,E1 21950.382,E2 21950.382} C_VEL
LIN {X 0,Y 449.281,Z 541.778,A -85,B 0,C 180,E1 21948.186,E2 21948.186} C_VEL
LIN {X 0,Y 449.922,Z 532.615,A -85,B 0,C 180,E1 21946.113,E2 21946.113} C_VEL
LIN {X 0,Y 450.71,Z 522.008,A -85,B 0,C 180,E1 21944.165,E2 21944.165} C_VEL
LIN {X 0,Y 451.64,Z 509.991,A -85,B 0,C 180,E1 21942.345,E2 21942.345} C_VEL
LIN {X 0,Y 452.666,Z 496.448,A -85,B 0,C 180,E1 21940.651,E2 21940.651} C_VEL
LIN {X 0,Y 453.757,Z 481.22,A -85,B 0,C 180,E1 21939.086,E2 21939.086} C_VEL
LIN {X 0,Y 454.81,Z 464.826,A -85,B 0,C 180,E1 21937.715,E2 21937.715} C_VEL
LIN {X 0,Y 455.737,Z 448.353,A -85,B 0,C 180,E1 21936.603,E2 21936.603} C_VEL
LIN {X 0,Y 456.609,Z 429.425,A -85,B 0,C 180,E1 21935.601,E2 21935.601} C_VEL
LIN {X 0,Y 457.263,Z 410.526,A -85,B 0,C 180,E1 21934.855,E2 21934.855} C_VEL
LIN {X 0,Y 457.707,Z 390.815,A -85,B 0,C 180,E1 21934.324,E2 21934.324} C_VEL
LIN {X 0,Y 460.063,Z 300.415,A -85,B 0,C 180,E1 21932.535,E2 21932.535} C_VEL
LIN {X 0,Y 464.144,Z 201.972,A -85,B 0,C 180,E1 21930.375,E2 21930.375} C_VEL
LIN {X 0,Y 464.087,Z 197.232,A -85,B 0,C 180,E1 21930.24,E2 21930.24} C_VEL
LIN {X 0,Y 463.303,Z 192.1,A -85,B 0,C 180,E1 21930.018,E2 21930.018} C_VEL
LIN {X 0,Y 464.638,Z 150.858,A -85,B 0,C 180,E1 21926.646,E2 21926.646} C_VEL
LIN {X 0,Y 464.418,Z 148.339,A -85,B 0,C 180,E1 21926.406,E2 21926.406} C_VEL
LIN {X 0,Y 460.818,Z 137.371,A -85,B 0,C 180,E1 21924.994,E2 21924.994} C_VEL
LIN {X 0,Y 456.332,Z 127.15,A -85,B 0,C 180,E1 21923.418,E2 21923.418} C_VEL
LIN {X 0,Y 454.067,Z 122.898,A -85,B 0,C 180,E1 21922.649,E2 21922.649} C_VEL
LIN {X 0,Y 452.15,Z 119.039,A -85,B 0,C 180,E1 21921.929,E2 21921.929} C_VEL
LIN {X 0,Y 449.693,Z 115.713,A -85,B 0,C 180,E1 21921.097,E2 21921.097} C_VEL
LIN {X 0,Y 449.087,Z 113.548,A -85,B 0,C 180,E1 21920.698,E2 21920.698} C_VEL
LIN {X 0,Y 449.087,Z 113.547,A -85,B 0,C 180,E1 21917.056,E2 21917.056} C_VEL
LIN {X 0,Y 449.104,Z 113.544,A -85,B 0,C 180,E1 21913.466,E2 21913.466} C_VEL
LIN {X 0,Y 449.078,Z 113.635,A -85,B 0,C 180,E1 21912.754,E2 21912.754} C_VEL
LIN {X 0,Y 450.49,Z 117.181,A -85,B 0,C 180,E1 21912.262,E2 21912.262} C_VEL
LIN {X 0,Y 458.212,Z 135.166,A -85,B 0,C 180,E1 21909.817,E2 21909.817} C_VEL
LIN {X 0,Y 466.195,Z 155.867,A -85,B 0,C 180,E1 21907.28,E2 21907.28} C_VEL
LIN {X 0,Y 465.689,Z 164.861,A -85,B 0,C 180,E1 21906.59,E2 21906.59} C_VEL
LIN {X 0,Y 468.759,Z 188.946,A -85,B 0,C 180,E1 21905.886,E2 21905.886} C_VEL
LIN {X 0,Y 463.824,Z 415.582,A -85,B 0,C 180,E1 21901.965,E2 21901.965} C_VEL
LIN {X 0,Y 462.879,Z 437.08,A -85,B 0,C 180,E1 21901.435,E2 21901.435} C_VEL
LIN {X 0,Y 461.682,Z 457.393,A -85,B 0,C 180,E1 21900.709,E2 21900.709} C_VEL
LIN {X 0,Y 460.276,Z 476.91,A -85,B 0,C 180,E1 21899.79,E2 21899.79} C_VEL
LIN {X 0,Y 458.648,Z 496.991,A -85,B 0,C 180,E1 21898.589,E2 21898.589} C_VEL
LIN {X 0,Y 456.882,Z 516.506,A -85,B 0,C 180,E1 21897.149,E2 21897.149} C_VEL
LIN {X 0,Y 455.162,Z 534.927,A -85,B 0,C 180,E1 21895.503,E2 21895.503} C_VEL
LIN {X 0,Y 453.569,Z 551.759,A -85,B 0,C 180,E1 21893.717,E2 21893.717} C_VEL
LIN {X 0,Y 452.161,Z 566.956,A -85,B 0,C 180,E1 21891.809,E2 21891.809} C_VEL
LIN {X 0,Y 450.962,Z 580.358,A -85,B 0,C 180,E1 21889.831,E2 21889.831} C_VEL
LIN {X 0,Y 449.968,Z 592.523,A -85,B 0,C 180,E1 21887.724,E2 21887.724} C_VEL
LIN {X 0,Y 449.175,Z 603.546,A -85,B 0,C 180,E1 21885.453,E2 21885.453} C_VEL
LIN {X 0,Y 448.587,Z 613.227,A -85,B 0,C 180,E1 21883.011,E2 21883.011} C_VEL
LIN {X 0,Y 448.251,Z 620.695,A -85,B 0,C 180,E1 21880.67,E2 21880.67} C_VEL
LIN {X 0,Y 448.057,Z 627.11,A -85,B 0,C 180,E1 21878.083,E2 21878.083} C_VEL
LIN {X 0,Y 447.974,Z 631.515,A -85,B 0,C 180,E1 21875.637,E2 21875.637} C_VEL
LIN {X 0,Y 447.956,Z 634.273,A -85,B 0,C 180,E1 21873.2,E2 21873.2} C_VEL
LIN {X 0,Y 447.958,Z 635.487,A -85,B 0,C 180,E1 21870.768,E2 21870.768} C_VEL
LIN {X 0,Y 447.954,Z 635.243,A -85,B 0,C 180,E1 21868.338,E2 21868.338} C_VEL
LIN {X 0,Y 447.96,Z 633.436,A -85,B 0,C 180,E1 21865.905,E2 21865.905} C_VEL
LIN {X 0,Y 447.987,Z 630.062,A -85,B 0,C 180,E1 21863.465,E2 21863.465} C_VEL
LIN {X 0,Y 448.117,Z 624.794,A -85,B 0,C 180,E1 21860.886,E2 21860.886} C_VEL
LIN {X 0,Y 448.36,Z 618.038,A -85,B 0,C 180,E1 21858.423,E2 21858.423} C_VEL
LIN {X 0,Y 448.808,Z 609.358,A -85,B 0,C 180,E1 21855.947,E2 21855.947} C_VEL
LIN {X 0,Y 449.479,Z 599.131,A -85,B 0,C 180,E1 21853.591,E2 21853.591} C_VEL
LIN {X 0,Y 450.374,Z 587.469,A -85,B 0,C 180,E1 21851.357,E2 21851.357} C_VEL
LIN {X 0,Y 451.567,Z 573.509,A -85,B 0,C 180,E1 21849.116,E2 21849.116} C_VEL
LIN {X 0,Y 452.96,Z 558.328,A -85,B 0,C 180,E1 21847.071,E2 21847.071} C_VEL
LIN {X 0,Y 454.477,Z 542.083,A -85,B 0,C 180,E1 21845.223,E2 21845.223} C_VEL
LIN {X 0,Y 456.133,Z 524.498,A -85,B 0,C 180,E1 21843.532,E2 21843.532} C_VEL
LIN {X 0,Y 457.839,Z 505.952,A -85,B 0,C 180,E1 21842.039,E2 21842.039} C_VEL
LIN {X 0,Y 459.515,Z 486.568,A -85,B 0,C 180,E1 21840.754,E2 21840.754} C_VEL
LIN {X 0,Y 461.108,Z 465.768,A -85,B 0,C 180,E1 21839.654,E2 21839.654} C_VEL
LIN {X 0,Y 462.494,Z 444.617,A -85,B 0,C 180,E1 21838.805,E2 21838.805} C_VEL
LIN {X 0,Y 463.533,Z 423.635,A -85,B 0,C 180,E1 21838.204,E2 21838.204} C_VEL
LIN {X 0,Y 464.496,Z 384.987,A -85,B 0,C 180,E1 21837.497,E2 21837.497} C_VEL
LIN {X 0,Y 468.699,Z 186.967,A -85,B 0,C 180,E1 21834.073,E2 21834.073} C_VEL
LIN {X 0,Y 465.634,Z 163.624,A -85,B 0,C 180,E1 21833.349,E2 21833.349} C_VEL
LIN {X 0,Y 466.167,Z 155.832,A -85,B 0,C 180,E1 21832.725,E2 21832.725} C_VEL
LIN {X 0,Y 458.528,Z 135.966,A -85,B 0,C 180,E1 21830.291,E2 21830.291} C_VEL
LIN {X 0,Y 450.475,Z 117.109,A -85,B 0,C 180,E1 21827.739,E2 21827.739} C_VEL
LIN {X 0,Y 449.083,Z 113.547,A -85,B 0,C 180,E1 21827.231,E2 21827.231} C_VEL
LIN {X 0,Y 449.1,Z 113.535,A -85,B 0,C 180,E1 21823.643,E2 21823.643} C_VEL
LIN {X 0,Y 449.126,Z 113.508,A -85,B 0,C 180,E1 21820.021,E2 21820.021} C_VEL
LIN {X 0,Y 449.12,Z 113.525,A -85,B 0,C 180,E1 21816.304,E2 21816.304} C_VEL
LIN {X 0,Y 449.103,Z 113.529,A -85,B 0,C 180,E1 21812.6,E2 21812.6} C_VEL
LIN {X 0,Y 449.08,Z 113.533,A -85,B 0,C 180,E1 21809.036,E2 21809.036} C_VEL
LIN {X 0,Y 449.078,Z 113.54,A -85,B 0,C 180,E1 21805.308,E2 21805.308} C_VEL
LIN {X 0,Y 449.088,Z 113.544,A -85,B 0,C 180,E1 21801.69,E2 21801.69} C_VEL
LIN {X 0,Y 449.112,Z 113.527,A -85,B 0,C 180,E1 21798.083,E2 21798.083} C_VEL
LIN {X 0,Y 449.133,Z 113.527,A -85,B 0,C 180,E1 21794.306,E2 21794.306} C_VEL
LIN {X 0,Y 449.115,Z 113.541,A -85,B 0,C 180,E1 21790.518,E2 21790.518} C_VEL
LIN {X 0,Y 449.085,Z 113.522,A -85,B 0,C 180,E1 21786.905,E2 21786.905} C_VEL
LIN {X 0,Y 449.073,Z 113.543,A -85,B 0,C 180,E1 21783.318,E2 21783.318} C_VEL
LIN {X 0,Y 449.072,Z 113.538,A -85,B 0,C 180,E1 21779.617,E2 21779.617} C_VEL
LIN {X 0,Y 449.089,Z 113.533,A -85,B 0,C 180,E1 21776.042,E2 21776.042} C_VEL
LIN {X 0,Y 449.115,Z 113.54,A -85,B 0,C 180,E1 21772.323,E2 21772.323} C_VEL
LIN {X 0,Y 449.114,Z 113.523,A -85,B 0,C 180,E1 21768.572,E2 21768.572} C_VEL
LIN {X 0,Y 449.094,Z 113.545,A -85,B 0,C 180,E1 21764.901,E2 21764.901} C_VEL
LIN {X 0,Y 449.071,Z 113.534,A -85,B 0,C 180,E1 21761.299,E2 21761.299} C_VEL
LIN {X 0,Y 449.062,Z 113.535,A -85,B 0,C 180,E1 21757.62,E2 21757.62} C_VEL
LIN {X 0,Y 449.075,Z 113.543,A -85,B 0,C 180,E1 21753.984,E2 21753.984} C_VEL
LIN {X 0,Y 449.097,Z 113.534,A -85,B 0,C 180,E1 21750.379,E2 21750.379} C_VEL
LIN {X 0,Y 449.106,Z 113.529,A -85,B 0,C 180,E1 21746.792,E2 21746.792} C_VEL
LIN {X 0,Y 449.076,Z 113.538,A -85,B 0,C 180,E1 21743.207,E2 21743.207} C_VEL
LIN {X 0,Y 449.062,Z 113.543,A -85,B 0,C 180,E1 21739.593,E2 21739.593} C_VEL
LIN {X 0,Y 449.059,Z 113.538,A -85,B 0,C 180,E1 21735.802,E2 21735.802} C_VEL
LIN {X 0,Y 449.066,Z 113.545,A -85,B 0,C 180,E1 21732.08,E2 21732.08} C_VEL
LIN {X 0,Y 449.14,Z 113.754,A -85,B 0,C 180,E1 21728.649,E2 21728.649} C_VEL
LIN {X 0,Y 456.813,Z 133.642,A -85,B 0,C 180,E1 21725.605,E2 21725.605} C_VEL
LIN {X 0,Y 463.411,Z 152.566,A -85,B 0,C 180,E1 21722.954,E2 21722.954} C_VEL
LIN {X 0,Y 461.875,Z 174.157,A -85,B 0,C 180,E1 21720.899,E2 21720.899} C_VEL
LIN {X 0,Y 466.483,Z 200.839,A -85,B 0,C 180,E1 21720.066,E2 21720.066} C_VEL
LIN {X 0,Y 465.37,Z 282.05,A -85,B 0,C 180,E1 21718.821,E2 21718.821} C_VEL
LIN {X 0,Y 464.433,Z 289.748,A -85,B 0,C 180,E1 21718.768,E2 21718.768} C_VEL
LIN {X 0,Y 458.801,Z 310.23,A -85,B 0,C 180,E1 21718.868,E2 21718.868} C_VEL
LIN {X 0,Y 458.084,Z 316.838,A -85,B 0,C 180,E1 21718.816,E2 21718.816} C_VEL
LIN {X 0,Y 457.054,Z 390.813,A -85,B 0,C 180,E1 21717.656,E2 21717.656} C_VEL
LIN {X 0,Y 456.303,Z 409.757,A -85,B 0,C 180,E1 21717.13,E2 21717.13} C_VEL
LIN {X 0,Y 455.237,Z 427.58,A -85,B 0,C 180,E1 21716.407,E2 21716.407} C_VEL
LIN {X 0,Y 453.805,Z 445.326,A -85,B 0,C 180,E1 21715.444,E2 21715.444} C_VEL
LIN {X 0,Y 452.159,Z 462.033,A -85,B 0,C 180,E1 21714.286,E2 21714.286} C_VEL
LIN {X 0,Y 450.387,Z 477.788,A -85,B 0,C 180,E1 21712.929,E2 21712.929} C_VEL
LIN {X 0,Y 448.459,Z 493.116,A -85,B 0,C 180,E1 21711.309,E2 21711.309} C_VEL
LIN {X 0,Y 446.613,Z 506.999,A -85,B 0,C 180,E1 21709.521,E2 21709.521} C_VEL
LIN {X 0,Y 444.994,Z 518.987,A -85,B 0,C 180,E1 21707.657,E2 21707.657} C_VEL
LIN {X 0,Y 443.518,Z 530.092,A -85,B 0,C 180,E1 21705.56,E2 21705.56} C_VEL
LIN {X 0,Y 442.324,Z 539.704,A -85,B 0,C 180,E1 21703.33,E2 21703.33} C_VEL
LIN {X 0,Y 441.413,Z 547.81,A -85,B 0,C 180,E1 21700.968,E2 21700.968} C_VEL
LIN {X 0,Y 440.804,Z 554.278,A -85,B 0,C 180,E1 21698.518,E2 21698.518} C_VEL
LIN {X 0,Y 440.434,Z 559.095,A -85,B 0,C 180,E1 21695.993,E2 21695.993} C_VEL
LIN {X 0,Y 440.25,Z 562.139,A -85,B 0,C 180,E1 21693.515,E2 21693.515} C_VEL
LIN {X 0,Y 440.185,Z 563.596,A -85,B 0,C 180,E1 21691.04,E2 21691.04} C_VEL
LIN {X 0,Y 440.19,Z 563.513,A -85,B 0,C 180,E1 21688.567,E2 21688.567} C_VEL
LIN {X 0,Y 440.275,Z 561.735,A -85,B 0,C 180,E1 21685.962,E2 21685.962} C_VEL
LIN {X 0,Y 440.485,Z 558.41,A -85,B 0,C 180,E1 21683.482,E2 21683.482} C_VEL
LIN {X 0,Y 440.885,Z 553.366,A -85,B 0,C 180,E1 21680.996,E2 21680.996} C_VEL
LIN {X 0,Y 441.514,Z 546.879,A -85,B 0,C 180,E1 21678.636,E2 21678.636} C_VEL
LIN {X 0,Y 442.467,Z 538.501,A -85,B 0,C 180,E1 21676.274,E2 21676.274} C_VEL
LIN {X 0,Y 443.71,Z 528.59,A -85,B 0,C 180,E1 21674.042,E2 21674.042} C_VEL
LIN {X 0,Y 445.237,Z 517.144,A -85,B 0,C 180,E1 21671.946,E2 21671.946} C_VEL
LIN {X 0,Y 446.94,Z 504.578,A -85,B 0,C 180,E1 21670.052,E2 21670.052} C_VEL
LIN {X 0,Y 448.725,Z 491.027,A -85,B 0,C 180,E1 21668.359,E2 21668.359} C_VEL
LIN {X 0,Y 450.607,Z 475.908,A -85,B 0,C 180,E1 21666.805,E2 21666.805} C_VEL
LIN {X 0,Y 452.321,Z 460.608,A -85,B 0,C 180,E1 21665.513,E2 21665.513} C_VEL
LIN {X 0,Y 453.885,Z 444.646,A -85,B 0,C 180,E1 21664.42,E2 21664.42} C_VEL
LIN {X 0,Y 455.32,Z 426.656,A -85,B 0,C 180,E1 21663.456,E2 21663.456} C_VEL
LIN {X 0,Y 456.405,Z 407.934,A -85,B 0,C 180,E1 21662.715,E2 21662.715} C_VEL
LIN {X 0,Y 457.124,Z 388.85,A -85,B 0,C 180,E1 21662.209,E2 21662.209} C_VEL
LIN {X 0,Y 459.678,Z 200.389,A -85,B 0,C 180,E1 21659.275,E2 21659.275} C_VEL
LIN {X 0,Y 454.863,Z 173.362,A -85,B 0,C 180,E1 21658.381,E2 21658.381} C_VEL
LIN {X 0,Y 456.238,Z 155.43,A -85,B 0,C 180,E1 21656.614,E2 21656.614} C_VEL
LIN {X 0,Y 449.905,Z 137.062,A -85,B 0,C 180,E1 21653.994,E2 21653.994} C_VEL
LIN {X 0,Y 443.564,Z 120.836,A -85,B 0,C 180,E1 21651.462,E2 21651.462} C_VEL
LIN {X 0,Y 441.155,Z 114.495,A -85,B 0,C 180,E1 21650.408,E2 21650.408} C_VEL
LIN {X 0,Y 441.171,Z 114.522,A -85,B 0,C 180,E1 21646.629,E2 21646.629} C_VEL
LIN {X 0,Y 441.184,Z 114.521,A -85,B 0,C 180,E1 21642.836,E2 21642.836} C_VEL
LIN {X 0,Y 441.192,Z 114.526,A -85,B 0,C 180,E1 21639.052,E2 21639.052} C_VEL
LIN {X 0,Y 441.227,Z 114.757,A -85,B 0,C 180,E1 21637.092,E2 21637.092} C_VEL
LIN {X 0,Y 450.473,Z 140.62,A -85,B 0,C 180,E1 21634.01,E2 21634.01} C_VEL
LIN {X 0,Y 453.657,Z 150.449,A -85,B 0,C 180,E1 21632.888,E2 21632.888} C_VEL
LIN {X 0,Y 452.455,Z 183.192,A -85,B 0,C 180,E1 21630.098,E2 21630.098} C_VEL
LIN {X 0,Y 454.889,Z 200.203,A -85,B 0,C 180,E1 21629.586,E2 21629.586} C_VEL
LIN {X 0,Y 450.403,Z 393.917,A -85,B 0,C 180,E1 21625.958,E2 21625.958} C_VEL
LIN {X 0,Y 449.757,Z 413.488,A -85,B 0,C 180,E1 21625.344,E2 21625.344} C_VEL
LIN {X 0,Y 448.896,Z 432.131,A -85,B 0,C 180,E1 21624.516,E2 21624.516} C_VEL
LIN {X 0,Y 447.871,Z 449.893,A -85,B 0,C 180,E1 21623.484,E2 21623.484} C_VEL
LIN {X 0,Y 446.73,Z 467.102,A -85,B 0,C 180,E1 21622.226,E2 21622.226} C_VEL
LIN {X 0,Y 445.543,Z 483.289,A -85,B 0,C 180,E1 21620.768,E2 21620.768} C_VEL
LIN {X 0,Y 444.41,Z 497.834,A -85,B 0,C 180,E1 21619.177,E2 21619.177} C_VEL
LIN {X 0,Y 443.367,Z 510.943,A -85,B 0,C 180,E1 21617.454,E2 21617.454} C_VEL
LIN {X 0,Y 442.448,Z 522.71,A -85,B 0,C 180,E1 21615.6,E2 21615.6} C_VEL
LIN {X 0,Y 441.689,Z 533.154,A -85,B 0,C 180,E1 21613.617,E2 21613.617} C_VEL
LIN {X 0,Y 441.091,Z 542.244,A -85,B 0,C 180,E1 21611.507,E2 21611.507} C_VEL
LIN {X 0,Y 440.664,Z 550.006,A -85,B 0,C 180,E1 21609.243,E2 21609.243} C_VEL
LIN {X 0,Y 440.403,Z 556.092,A -85,B 0,C 180,E1 21606.911,E2 21606.911} C_VEL
LIN {X 0,Y 440.254,Z 560.419,A -85,B 0,C 180,E1 21604.559,E2 21604.559} C_VEL
LIN {X 0,Y 440.204,Z 563.026,A -85,B 0,C 180,E1 21602.213,E2 21602.213} C_VEL
LIN {X 0,Y 440.204,Z 563.985,A -85,B 0,C 180,E1 21599.87,E2 21599.87} C_VEL
LIN {X 0,Y 440.237,Z 563.299,A -85,B 0,C 180,E1 21597.527,E2 21597.527} C_VEL
LIN {X 0,Y 440.335,Z 560.957,A -85,B 0,C 180,E1 21595.181,E2 21595.181} C_VEL
LIN {X 0,Y 440.531,Z 556.889,A -85,B 0,C 180,E1 21592.829,E2 21592.829} C_VEL
LIN {X 0,Y 440.84,Z 551.356,A -85,B 0,C 180,E1 21590.602,E2 21590.602} C_VEL
LIN {X 0,Y 441.323,Z 543.989,A -85,B 0,C 180,E1 21588.368,E2 21588.368} C_VEL
LIN {X 0,Y 442.031,Z 534.556,A -85,B 0,C 180,E1 21586.127,E2 21586.127} C_VEL
LIN {X 0,Y 442.925,Z 523.452,A -85,B 0,C 180,E1 21584.014,E2 21584.014} C_VEL
LIN {X 0,Y 443.907,Z 511.513,A -85,B 0,C 180,E1 21582.162,E2 21582.162} C_VEL
LIN {X 0,Y 445,Z 498.145,A -85,B 0,C 180,E1 21580.441,E2 21580.441} C_VEL
LIN {X 0,Y 446.163,Z 483.147,A -85,B 0,C 180,E1 21578.851,E2 21578.851} C_VEL
LIN {X 0,Y 447.281,Z 467.003,A -85,B 0,C 180,E1 21577.457,E2 21577.457} C_VEL
LIN {X 0,Y 448.332,Z 449.848,A -85,B 0,C 180,E1 21576.263,E2 21576.263} C_VEL
LIN {X 0,Y 449.244,Z 431.567,A -85,B 0,C 180,E1 21575.265,E2 21575.265} C_VEL
LIN {X 0,Y 449.986,Z 411.866,A -85,B 0,C 180,E1 21574.461,E2 21574.461} C_VEL
LIN {X 0,Y 450.487,Z 392.216,A -85,B 0,C 180,E1 21573.909,E2 21573.909} C_VEL
LIN {X 0,Y 452.96,Z 307.138,A -85,B 0,C 180,E1 21572.161,E2 21572.161} C_VEL
LIN {X 0,Y 457.411,Z 209.209,A -85,B 0,C 180,E1 21569.935,E2 21569.935} C_VEL
LIN {X 0,Y 457.759,Z 199.089,A -85,B 0,C 180,E1 21569.673,E2 21569.673} C_VEL
LIN {X 0,Y 456.917,Z 193.454,A -85,B 0,C 180,E1 21569.418,E2 21569.418} C_VEL
LIN {X 0,Y 458.489,Z 152.852,A -85,B 0,C 180,E1 21566.045,E2 21566.045} C_VEL
LIN {X 0,Y 455.102,Z 142.072,A -85,B 0,C 180,E1 21564.597,E2 21564.597} C_VEL
LIN {X 0,Y 451.22,Z 132.882,A -85,B 0,C 180,E1 21563.125,E2 21563.125} C_VEL
LIN {X 0,Y 448.879,Z 128.402,A -85,B 0,C 180,E1 21562.256,E2 21562.256} C_VEL
LIN {X 0,Y 447.054,Z 124.776,A -85,B 0,C 180,E1 21561.518,E2 21561.518} C_VEL
LIN {X 0,Y 444.909,Z 121.12,A -85,B 0,C 180,E1 21560.632,E2 21560.632} C_VEL
LIN {X 0,Y 444.668,Z 120.226,A -85,B 0,C 180,E1 21560.467,E2 21560.467} C_VEL
LIN {X 0,Y 441.962,Z 117.119,A -85,B 0,C 180,E1 21559.342,E2 21559.342} C_VEL
LIN {X 0,Y 441.142,Z 114.536,A -85,B 0,C 180,E1 21558.674,E2 21558.674} C_VEL
LIN {X 0,Y 441.141,Z 114.536,A -85,B 0,C 180,E1 21554.996,E2 21554.996} C_VEL
LIN {X 0,Y 441.176,Z 114.575,A -85,B 0,C 180,E1 21553.549,E2 21553.549} C_VEL
LIN {X 0,Y 442.308,Z 117.811,A -85,B 0,C 180,E1 21553.101,E2 21553.101} C_VEL
LIN {X 0,Y 449.33,Z 133.619,A -85,B 0,C 180,E1 21550.837,E2 21550.837} C_VEL
LIN {X 0,Y 457.232,Z 153.494,A -85,B 0,C 180,E1 21548.275,E2 21548.275} C_VEL
LIN {X 0,Y 459.202,Z 159.517,A -85,B 0,C 180,E1 21547.566,E2 21547.566} C_VEL
LIN {X 0,Y 458.873,Z 165.002,A -85,B 0,C 180,E1 21547.157,E2 21547.157} C_VEL
LIN {X 0,Y 462.032,Z 190.166,A -85,B 0,C 180,E1 21546.406,E2 21546.406} C_VEL
LIN {X 0,Y 456.842,Z 414.589,A -85,B 0,C 180,E1 21542.467,E2 21542.467} C_VEL
LIN {X 0,Y 455.881,Z 435.746,A -85,B 0,C 180,E1 21541.947,E2 21541.947} C_VEL
LIN {X 0,Y 454.634,Z 455.926,A -85,B 0,C 180,E1 21541.227,E2 21541.227} C_VEL
LIN {X 0,Y 453.111,Z 475.926,A -85,B 0,C 180,E1 21540.28,E2 21540.28} C_VEL
LIN {X 0,Y 451.407,Z 495.545,A -85,B 0,C 180,E1 21539.095,E2 21539.095} C_VEL
LIN {X 0,Y 449.578,Z 514.36,A -85,B 0,C 180,E1 21537.699,E2 21537.699} C_VEL
LIN {X 0,Y 447.804,Z 532.26,A -85,B 0,C 180,E1 21536.096,E2 21536.096} C_VEL
LIN {X 0,Y 446.072,Z 549.232,A -85,B 0,C 180,E1 21534.288,E2 21534.288} C_VEL
LIN {X 0,Y 444.507,Z 564.969,A -85,B 0,C 180,E1 21532.307,E2 21532.307} C_VEL
LIN {X 0,Y 443.15,Z 579.299,A -85,B 0,C 180,E1 21530.183,E2 21530.183} C_VEL
LIN {X 0,Y 442.1,Z 591.496,A -85,B 0,C 180,E1 21528.05,E2 21528.05} C_VEL
LIN {X 0,Y 441.226,Z 603.006,A -85,B 0,C 180,E1 21525.645,E2 21525.645} C_VEL
LIN {X 0,Y 440.624,Z 612.453,A -85,B 0,C 180,E1 21523.225,E2 21523.225} C_VEL
LIN {X 0,Y 440.276,Z 619.908,A -85,B 0,C 180,E1 21520.866,E2 21520.866} C_VEL
LIN {X 0,Y 440.073,Z 626.395,A -85,B 0,C 180,E1 21518.23,E2 21518.23} C_VEL
LIN {X 0,Y 439.992,Z 630.84,A -85,B 0,C 180,E1 21515.739,E2 21515.739} C_VEL
LIN {X 0,Y 439.978,Z 633.617,A -85,B 0,C 180,E1 21513.258,E2 21513.258} C_VEL
LIN {X 0,Y 439.985,Z 634.842,A -85,B 0,C 180,E1 21510.782,E2 21510.782} C_VEL
LIN {X 0,Y 439.98,Z 634.594,A -85,B 0,C 180,E1 21508.308,E2 21508.308} C_VEL
LIN {X 0,Y 439.979,Z 632.775,A -85,B 0,C 180,E1 21505.831,E2 21505.831} C_VEL
LIN {X 0,Y 440.008,Z 629.371,A -85,B 0,C 180,E1 21503.346,E2 21503.346} C_VEL
LIN {X 0,Y 440.138,Z 624.052,A -85,B 0,C 180,E1 21500.719,E2 21500.719} C_VEL
LIN {X 0,Y 440.391,Z 617.222,A -85,B 0,C 180,E1 21498.21,E2 21498.21} C_VEL
LIN {X 0,Y 440.864,Z 608.475,A -85,B 0,C 180,E1 21495.689,E2 21495.689} C_VEL
LIN {X 0,Y 441.576,Z 598.154,A -85,B 0,C 180,E1 21493.289,E2 21493.289} C_VEL
LIN {X 0,Y 442.533,Z 586.382,A -85,B 0,C 180,E1 21491.014,E2 21491.014} C_VEL
LIN {X 0,Y 443.719,Z 573.195,A -85,B 0,C 180,E1 21488.868,E2 21488.868} C_VEL
LIN {X 0,Y 445.237,Z 557.563,A -85,B 0,C 180,E1 21486.72,E2 21486.72} C_VEL
LIN {X 0,Y 446.867,Z 541.44,A -85,B 0,C 180,E1 21484.843,E2 21484.843} C_VEL
LIN {X 0,Y 448.565,Z 524.728,A -85,B 0,C 180,E1 21483.191,E2 21483.191} C_VEL
LIN {X 0,Y 450.338,Z 506.812,A -85,B 0,C 180,E1 21481.705,E2 21481.705} C_VEL
LIN {X 0,Y 452.195,Z 486.701,A -85,B 0,C 180,E1 21480.339,E2 21480.339} C_VEL
LIN {X 0,Y 453.818,Z 466.823,A -85,B 0,C 180,E1 21479.261,E2 21479.261} C_VEL
LIN {X 0,Y 455.237,Z 446.675,A -85,B 0,C 180,E1 21478.417,E2 21478.417} C_VEL
LIN {X 0,Y 456.392,Z 425.892,A -85,B 0,C 180,E1 21477.785,E2 21477.785} C_VEL
LIN {X 0,Y 457.258,Z 397.239,A -85,B 0,C 180,E1 21477.22,E2 21477.22} C_VEL
LIN {X 0,Y 462.02,Z 188.504,A -85,B 0,C 180,E1 21473.562,E2 21473.562} C_VEL
LIN {X 0,Y 458.803,Z 163.859,A -85,B 0,C 180,E1 21472.79,E2 21472.79} C_VEL
LIN {X 0,Y 459.048,Z 158.584,A -85,B 0,C 180,E1 21472.349,E2 21472.349} C_VEL
LIN {X 0,Y 451.377,Z 138.627,A -85,B 0,C 180,E1 21469.837,E2 21469.837} C_VEL
LIN {X 0,Y 444.293,Z 121.991,A -85,B 0,C 180,E1 21467.537,E2 21467.537} C_VEL
LIN {X 0,Y 441.278,Z 115.2,A -85,B 0,C 180,E1 21466.533,E2 21466.533} C_VEL
LIN {X 0,Y 441.172,Z 114.526,A -85,B 0,C 180,E1 21466.452,E2 21466.452} C_VEL
LIN {X 0,Y 441.147,Z 114.524,A -85,B 0,C 180,E1 21462.839,E2 21462.839} C_VEL
LIN {X 0,Y 441.135,Z 114.486,A -85,B 0,C 180,E1 21459.182,E2 21459.182} C_VEL
LIN {X 0,Y 441.147,Z 114.534,A -85,B 0,C 180,E1 21455.466,E2 21455.466} C_VEL
LIN {X 0,Y 441.163,Z 114.527,A -85,B 0,C 180,E1 21451.801,E2 21451.801} C_VEL
LIN {X 0,Y 441.19,Z 114.516,A -85,B 0,C 180,E1 21448.124,E2 21448.124} C_VEL
LIN {X 0,Y 441.184,Z 114.515,A -85,B 0,C 180,E1 21444.351,E2 21444.351} C_VEL
LIN {X 0,Y 441.16,Z 114.532,A -85,B 0,C 180,E1 21440.705,E2 21440.705} C_VEL
LIN {X 0,Y 441.143,Z 114.528,A -85,B 0,C 180,E1 21437,E2 21437} C_VEL
LIN {X 0,Y 441.133,Z 114.513,A -85,B 0,C 180,E1 21433.367,E2 21433.367} C_VEL
LIN {X 0,Y 441.138,Z 114.532,A -85,B 0,C 180,E1 21429.624,E2 21429.624} C_VEL
LIN {X 0,Y 441.156,Z 114.519,A -85,B 0,C 180,E1 21425.984,E2 21425.984} C_VEL
LIN {X 0,Y 441.177,Z 114.518,A -85,B 0,C 180,E1 21422.338,E2 21422.338} C_VEL
LIN {X 0,Y 441.178,Z 114.527,A -85,B 0,C 180,E1 21418.571,E2 21418.571} C_VEL
LIN {X 0,Y 441.157,Z 114.512,A -85,B 0,C 180,E1 21414.798,E2 21414.798} C_VEL
LIN {X 0,Y 441.138,Z 114.533,A -85,B 0,C 180,E1 21411.187,E2 21411.187} C_VEL
LIN {X 0,Y 441.13,Z 114.522,A -85,B 0,C 180,E1 21407.432,E2 21407.432} C_VEL
LIN {X 0,Y 441.129,Z 114.526,A -85,B 0,C 180,E1 21403.676,E2 21403.676} C_VEL
LIN {X 0,Y 441.139,Z 114.534,A -85,B 0,C 180,E1 21399.986,E2 21399.986} C_VEL
LIN {X 0,Y 441.16,Z 114.514,A -85,B 0,C 180,E1 21396.349,E2 21396.349} C_VEL
LIN {X 0,Y 441.178,Z 114.516,A -85,B 0,C 180,E1 21392.608,E2 21392.608} C_VEL
LIN {X 0,Y 441.163,Z 114.533,A -85,B 0,C 180,E1 21388.886,E2 21388.886} C_VEL
LIN {X 0,Y 441.145,Z 114.532,A -85,B 0,C 180,E1 21385.131,E2 21385.131} C_VEL
LIN {X 0,Y 441.128,Z 114.533,A -85,B 0,C 180,E1 21381.44,E2 21381.44} C_VEL
LIN {X 0,Y 441.123,Z 114.536,A -85,B 0,C 180,E1 21377.831,E2 21377.831} C_VEL
LIN {X 0,Y 441.129,Z 114.537,A -85,B 0,C 180,E1 21374.068,E2 21374.068} C_VEL
LIN {X 0,Y 441.147,Z 114.528,A -85,B 0,C 180,E1 21370.399,E2 21370.399} C_VEL
LIN {X 0,Y 441.152,Z 114.695,A -85,B 0,C 180,E1 21369.434,E2 21369.434} C_VEL
LIN {X 0,Y 449.173,Z 135.167,A -85,B 0,C 180,E1 21366.192,E2 21366.192} C_VEL
LIN {X 0,Y 455.524,Z 153.308,A -85,B 0,C 180,E1 21363.581,E2 21363.581} C_VEL
LIN {X 0,Y 456.291,Z 156.088,A -85,B 0,C 180,E1 21363.216,E2 21363.216} C_VEL
LIN {X 0,Y 454.915,Z 174.027,A -85,B 0,C 180,E1 21361.491,E2 21361.491} C_VEL
LIN {X 0,Y 459.759,Z 202.154,A -85,B 0,C 180,E1 21360.589,E2 21360.589} C_VEL
LIN {X 0,Y 458.084,Z 316.838,A -85,B 0,C 180,E1 21358.816,E2 21358.816} C_VEL
LIN {X 0,Y 457.146,Z 324.534,A -85,B 0,C 180,E1 21358.763,E2 21358.763} C_VEL
LIN {X 0,Y 451.508,Z 345.011,A -85,B 0,C 180,E1 21358.866,E2 21358.866} C_VEL
LIN {X 0,Y 450.78,Z 351.618,A -85,B 0,C 180,E1 21358.814,E2 21358.814} C_VEL
LIN {X 0,Y 450.129,Z 391.933,A -85,B 0,C 180,E1 21358.149,E2 21358.149} C_VEL
LIN {X 0,Y 449.334,Z 410.656,A -85,B 0,C 180,E1 21357.614,E2 21357.614} C_VEL
LIN {X 0,Y 448.166,Z 428.848,A -85,B 0,C 180,E1 21356.857,E2 21356.857} C_VEL
LIN {X 0,Y 446.66,Z 446.408,A -85,B 0,C 180,E1 21355.88,E2 21355.88} C_VEL
LIN {X 0,Y 444.93,Z 462.998,A -85,B 0,C 180,E1 21354.706,E2 21354.706} C_VEL
LIN {X 0,Y 443.065,Z 478.677,A -85,B 0,C 180,E1 21353.33,E2 21353.33} C_VEL
LIN {X 0,Y 441.109,Z 493.406,A -85,B 0,C 180,E1 21351.752,E2 21351.752} C_VEL
LIN {X 0,Y 439.182,Z 507.125,A -85,B 0,C 180,E1 21349.967,E2 21349.967} C_VEL
LIN {X 0,Y 437.366,Z 519.736,A -85,B 0,C 180,E1 21347.975,E2 21347.975} C_VEL
LIN {X 0,Y 435.795,Z 530.815,A -85,B 0,C 180,E1 21345.843,E2 21345.843} C_VEL
LIN {X 0,Y 434.522,Z 540.405,A -85,B 0,C 180,E1 21343.573,E2 21343.573} C_VEL
LIN {X 0,Y 433.545,Z 548.494,A -85,B 0,C 180,E1 21341.169,E2 21341.169} C_VEL
LIN {X 0,Y 432.883,Z 554.969,A -85,B 0,C 180,E1 21338.665,E2 21338.665} C_VEL
LIN {X 0,Y 432.483,Z 559.752,A -85,B 0,C 180,E1 21336.104,E2 21336.104} C_VEL
LIN {X 0,Y 432.283,Z 562.788,A -85,B 0,C 180,E1 21333.58,E2 21333.58} C_VEL
LIN {X 0,Y 432.212,Z 564.241,A -85,B 0,C 180,E1 21331.06,E2 21331.06} C_VEL
LIN {X 0,Y 432.217,Z 564.158,A -85,B 0,C 180,E1 21328.541,E2 21328.541} C_VEL
LIN {X 0,Y 432.311,Z 562.386,A -85,B 0,C 180,E1 21325.888,E2 21325.888} C_VEL
LIN {X 0,Y 432.539,Z 559.071,A -85,B 0,C 180,E1 21323.362,E2 21323.362} C_VEL
LIN {X 0,Y 432.973,Z 554.039,A -85,B 0,C 180,E1 21320.831,E2 21320.831} C_VEL
LIN {X 0,Y 433.654,Z 547.568,A -85,B 0,C 180,E1 21318.428,E2 21318.428} C_VEL
LIN {X 0,Y 434.677,Z 539.209,A -85,B 0,C 180,E1 21316.023,E2 21316.023} C_VEL
LIN {X 0,Y 436.004,Z 529.321,A -85,B 0,C 180,E1 21313.752,E2 21313.752} C_VEL
LIN {X 0,Y 437.631,Z 517.904,A -85,B 0,C 180,E1 21311.621,E2 21311.621} C_VEL
LIN {X 0,Y 439.433,Z 505.374,A -85,B 0,C 180,E1 21309.696,E2 21309.696} C_VEL
LIN {X 0,Y 441.319,Z 491.872,A -85,B 0,C 180,E1 21307.977,E2 21307.977} C_VEL
LIN {X 0,Y 443.302,Z 476.819,A -85,B 0,C 180,E1 21306.399,E2 21306.399} C_VEL
LIN {X 0,Y 445.2,Z 460.731,A -85,B 0,C 180,E1 21305.024,E2 21305.024} C_VEL
LIN {X 0,Y 446.848,Z 444.685,A -85,B 0,C 180,E1 21303.915,E2 21303.915} C_VEL
LIN {X 0,Y 448.359,Z 426.557,A -85,B 0,C 180,E1 21302.939,E2 21302.939} C_VEL
LIN {X 0,Y 449.482,Z 408.141,A -85,B 0,C 180,E1 21302.204,E2 21302.204} C_VEL
LIN {X 0,Y 450.24,Z 389.087,A -85,B 0,C 180,E1 21301.695,E2 21301.695} C_VEL
LIN {X 0,Y 453.013,Z 201.79,A -85,B 0,C 180,E1 21298.738,E2 21298.738} C_VEL
LIN {X 0,Y 447.969,Z 173.163,A -85,B 0,C 180,E1 21297.761,E2 21297.761} C_VEL
LIN {X 0,Y 449.258,Z 158.871,A -85,B 0,C 180,E1 21296.343,E2 21296.343} C_VEL
LIN {X 0,Y 443.37,Z 141.522,A -85,B 0,C 180,E1 21293.837,E2 21293.837} C_VEL
LIN {X 0,Y 437.087,Z 125.289,A -85,B 0,C 180,E1 21291.266,E2 21291.266} C_VEL
LIN {X 0,Y 433.269,Z 115.578,A -85,B 0,C 180,E1 21289.641,E2 21289.641} C_VEL
LIN {X 0,Y 433.257,Z 115.513,A -85,B 0,C 180,E1 21285.817,E2 21285.817} C_VEL
LIN {X 0,Y 433.256,Z 115.518,A -85,B 0,C 180,E1 21282.003,E2 21282.003} C_VEL
LIN {X 0,Y 433.259,Z 115.52,A -85,B 0,C 180,E1 21278.206,E2 21278.206} C_VEL
LIN {X 0,Y 433.265,Z 115.634,A -85,B 0,C 180,E1 21277.668,E2 21277.668} C_VEL
LIN {X 0,Y 442.559,Z 141.393,A -85,B 0,C 180,E1 21274.547,E2 21274.547} C_VEL
LIN {X 0,Y 446.404,Z 153.374,A -85,B 0,C 180,E1 21273.171,E2 21273.171} C_VEL
LIN {X 0,Y 445.221,Z 183.577,A -85,B 0,C 180,E1 21270.574,E2 21270.574} C_VEL
LIN {X 0,Y 447.724,Z 201.252,A -85,B 0,C 180,E1 21270.028,E2 21270.028} C_VEL
LIN {X 0,Y 442.942,Z 394.496,A -85,B 0,C 180,E1 21266.322,E2 21266.322} C_VEL
LIN {X 0,Y 442.26,Z 414.072,A -85,B 0,C 180,E1 21265.695,E2 21265.695} C_VEL
LIN {X 0,Y 441.335,Z 433.073,A -85,B 0,C 180,E1 21264.833,E2 21264.833} C_VEL
LIN {X 0,Y 440.23,Z 451.258,A -85,B 0,C 180,E1 21263.75,E2 21263.75} C_VEL
LIN {X 0,Y 439.001,Z 468.857,A -85,B 0,C 180,E1 21262.427,E2 21262.427} C_VEL
LIN {X 0,Y 437.762,Z 484.927,A -85,B 0,C 180,E1 21260.937,E2 21260.937} C_VEL
LIN {X 0,Y 436.543,Z 499.844,A -85,B 0,C 180,E1 21259.258,E2 21259.258} C_VEL
LIN {X 0,Y 435.397,Z 513.683,A -85,B 0,C 180,E1 21257.37,E2 21257.37} C_VEL
LIN {X 0,Y 434.398,Z 525.959,A -85,B 0,C 180,E1 21255.329,E2 21255.329} C_VEL
LIN {X 0,Y 433.607,Z 536.472,A -85,B 0,C 180,E1 21253.196,E2 21253.196} C_VEL
LIN {X 0,Y 433.032,Z 545.063,A -85,B 0,C 180,E1 21251.049,E2 21251.049} C_VEL
LIN {X 0,Y 432.628,Z 552.26,A -85,B 0,C 180,E1 21248.774,E2 21248.774} C_VEL
LIN {X 0,Y 432.383,Z 557.963,A -85,B 0,C 180,E1 21246.373,E2 21246.373} C_VEL
LIN {X 0,Y 432.262,Z 561.862,A -85,B 0,C 180,E1 21243.979,E2 21243.979} C_VEL
LIN {X 0,Y 432.218,Z 564.06,A -85,B 0,C 180,E1 21241.591,E2 21241.591} C_VEL
LIN {X 0,Y 432.237,Z 564.606,A -85,B 0,C 180,E1 21239.205,E2 21239.205} C_VEL
LIN {X 0,Y 432.292,Z 563.501,A -85,B 0,C 180,E1 21236.818,E2 21236.818} C_VEL
LIN {X 0,Y 432.425,Z 560.716,A -85,B 0,C 180,E1 21234.427,E2 21234.427} C_VEL
LIN {X 0,Y 432.689,Z 556.163,A -85,B 0,C 180,E1 21232.031,E2 21232.031} C_VEL
LIN {X 0,Y 433.08,Z 550.127,A -85,B 0,C 180,E1 21229.76,E2 21229.76} C_VEL
LIN {X 0,Y 433.683,Z 542.215,A -85,B 0,C 180,E1 21227.484,E2 21227.484} C_VEL
LIN {X 0,Y 434.467,Z 532.77,A -85,B 0,C 180,E1 21225.336,E2 21225.336} C_VEL
LIN {X 0,Y 435.475,Z 521.246,A -85,B 0,C 180,E1 21223.226,E2 21223.226} C_VEL
LIN {X 0,Y 436.573,Z 508.868,A -85,B 0,C 180,E1 21221.368,E2 21221.368} C_VEL
LIN {X 0,Y 437.739,Z 495.265,A -85,B 0,C 180,E1 21219.685,E2 21219.685} C_VEL
LIN {X 0,Y 438.971,Z 480.171,A -85,B 0,C 180,E1 21218.136,E2 21218.136} C_VEL
LIN {X 0,Y 440.126,Z 464.266,A -85,B 0,C 180,E1 21216.804,E2 21216.804} C_VEL
LIN {X 0,Y 441.285,Z 446.008,A -85,B 0,C 180,E1 21215.575,E2 21215.575} C_VEL
LIN {X 0,Y 442.207,Z 427.964,A -85,B 0,C 180,E1 21214.63,E2 21214.63} C_VEL
LIN {X 0,Y 442.924,Z 408.675,A -85,B 0,C 180,E1 21213.889,E2 21213.889} C_VEL
LIN {X 0,Y 443.479,Z 386.763,A -85,B 0,C 180,E1 21213.324,E2 21213.324} C_VEL
LIN {X 0,Y 446.243,Z 305.891,A -85,B 0,C 180,E1 21211.586,E2 21211.586} C_VEL
LIN {X 0,Y 451.159,Z 210.051,A -85,B 0,C 180,E1 21209.314,E2 21209.314} C_VEL
LIN {X 0,Y 451.528,Z 200.6,A -85,B 0,C 180,E1 21209.057,E2 21209.057} C_VEL
LIN {X 0,Y 450.728,Z 194.21,A -85,B 0,C 180,E1 21208.729,E2 21208.729} C_VEL
LIN {X 0,Y 452.426,Z 156.396,A -85,B 0,C 180,E1 21205.521,E2 21205.521} C_VEL
LIN {X 0,Y 449.558,Z 146.975,A -85,B 0,C 180,E1 21204.202,E2 21204.202} C_VEL
LIN {X 0,Y 446.053,Z 138.269,A -85,B 0,C 180,E1 21202.728,E2 21202.728} C_VEL
LIN {X 0,Y 442.569,Z 131.05,A -85,B 0,C 180,E1 21201.209,E2 21201.209} C_VEL
LIN {X 0,Y 440.295,Z 126.767,A -85,B 0,C 180,E1 21200.136,E2 21200.136} C_VEL
LIN {X 0,Y 437.826,Z 123.116,A -85,B 0,C 180,E1 21198.875,E2 21198.875} C_VEL
LIN {X 0,Y 437.227,Z 121.511,A -85,B 0,C 180,E1 21198.4,E2 21198.4} C_VEL
LIN {X 0,Y 434.432,Z 118.896,A -85,B 0,C 180,E1 21196.468,E2 21196.468} C_VEL
LIN {X 0,Y 433.588,Z 117.183,A -85,B 0,C 180,E1 21194.882,E2 21194.882} C_VEL
LIN {X 0,Y 433.522,Z 116.952,A -85,B 0,C 180,E1 21194.206,E2 21194.206} C_VEL
LIN {X 0,Y 437.013,Z 124.581,A -85,B 0,C 180,E1 21193.03,E2 21193.03} C_VEL
LIN {X 0,Y 444.176,Z 141.14,A -85,B 0,C 180,E1 21190.659,E2 21190.659} C_VEL
LIN {X 0,Y 451.573,Z 160.225,A -85,B 0,C 180,E1 21188.184,E2 21188.184} C_VEL
LIN {X 0,Y 452.193,Z 162.398,A -85,B 0,C 180,E1 21187.93,E2 21187.93} C_VEL
LIN {X 0,Y 452.113,Z 165.268,A -85,B 0,C 180,E1 21187.738,E2 21187.738} C_VEL
LIN {X 0,Y 455.342,Z 191.385,A -85,B 0,C 180,E1 21186.942,E2 21186.942} C_VEL
LIN {X 0,Y 449.903,Z 413.735,A -85,B 0,C 180,E1 21182.983,E2 21182.983} C_VEL
LIN {X 0,Y 448.927,Z 434.649,A -85,B 0,C 180,E1 21182.469,E2 21182.469} C_VEL
LIN {X 0,Y 447.595,Z 455.002,A -85,B 0,C 180,E1 21181.741,E2 21181.741} C_VEL
LIN {X 0,Y 445.985,Z 475.061,A -85,B 0,C 180,E1 21180.783,E2 21180.783} C_VEL
LIN {X 0,Y 444.109,Z 495.33,A -85,B 0,C 180,E1 21179.542,E2 21179.542} C_VEL
LIN {X 0,Y 442.18,Z 513.99,A -85,B 0,C 180,E1 21178.132,E2 21178.132} C_VEL
LIN {X 0,Y 440.327,Z 531.51,A -85,B 0,C 180,E1 21176.535,E2 21176.535} C_VEL
LIN {X 0,Y 438.491,Z 548.268,A -85,B 0,C 180,E1 21174.723,E2 21174.723} C_VEL
LIN {X 0,Y 436.814,Z 563.971,A -85,B 0,C 180,E1 21172.712,E2 21172.712} C_VEL
LIN {X 0,Y 435.376,Z 578.15,A -85,B 0,C 180,E1 21170.572,E2 21170.572} C_VEL
LIN {X 0,Y 434.182,Z 591.15,A -85,B 0,C 180,E1 21168.252,E2 21168.252} C_VEL
LIN {X 0,Y 433.314,Z 602.062,A -85,B 0,C 180,E1 21165.938,E2 21165.938} C_VEL
LIN {X 0,Y 432.675,Z 611.5,A -85,B 0,C 180,E1 21163.498,E2 21163.498} C_VEL
LIN {X 0,Y 432.302,Z 619.115,A -85,B 0,C 180,E1 21161.068,E2 21161.068} C_VEL
LIN {X 0,Y 432.09,Z 625.392,A -85,B 0,C 180,E1 21158.517,E2 21158.517} C_VEL
LIN {X 0,Y 432.009,Z 629.978,A -85,B 0,C 180,E1 21155.979,E2 21155.979} C_VEL
LIN {X 0,Y 432.001,Z 632.832,A -85,B 0,C 180,E1 21153.451,E2 21153.451} C_VEL
LIN {X 0,Y 432.011,Z 634.196,A -85,B 0,C 180,E1 21150.797,E2 21150.797} C_VEL
LIN {X 0,Y 432.006,Z 633.944,A -85,B 0,C 180,E1 21148.277,E2 21148.277} C_VEL
LIN {X 0,Y 431.998,Z 632.111,A -85,B 0,C 180,E1 21145.753,E2 21145.753} C_VEL
LIN {X 0,Y 432.037,Z 628.529,A -85,B 0,C 180,E1 21143.132,E2 21143.132} C_VEL
LIN {X 0,Y 432.157,Z 623.305,A -85,B 0,C 180,E1 21140.546,E2 21140.546} C_VEL
LIN {X 0,Y 432.422,Z 616.368,A -85,B 0,C 180,E1 21137.979,E2 21137.979} C_VEL
LIN {X 0,Y 432.933,Z 607.47,A -85,B 0,C 180,E1 21135.392,E2 21135.392} C_VEL
LIN {X 0,Y 433.682,Z 597.176,A -85,B 0,C 180,E1 21132.975,E2 21132.975} C_VEL
LIN {X 0,Y 434.705,Z 585.315,A -85,B 0,C 180,E1 21130.659,E2 21130.659} C_VEL
LIN {X 0,Y 435.974,Z 572.111,A -85,B 0,C 180,E1 21128.474,E2 21128.474} C_VEL
LIN {X 0,Y 437.604,Z 556.5,A -85,B 0,C 180,E1 21126.289,E2 21126.289} C_VEL
LIN {X 0,Y 439.454,Z 539.468,A -85,B 0,C 180,E1 21124.288,E2 21124.288} C_VEL
LIN {X 0,Y 441.363,Z 521.811,A -85,B 0,C 180,E1 21122.549,E2 21122.549} C_VEL
LIN {X 0,Y 443.222,Z 503.946,A -85,B 0,C 180,E1 21121.078,E2 21121.078} C_VEL
LIN {X 0,Y 445.09,Z 484.942,A -85,B 0,C 180,E1 21119.789,E2 21119.789} C_VEL
LIN {X 0,Y 446.84,Z 464.683,A -85,B 0,C 180,E1 21118.69,E2 21118.69} C_VEL
LIN {X 0,Y 448.41,Z 443.459,A -85,B 0,C 180,E1 21117.817,E2 21117.817} C_VEL
LIN {X 0,Y 449.581,Z 422.173,A -85,B 0,C 180,E1 21117.196,E2 21117.196} C_VEL
LIN {X 0,Y 450.928,Z 371.204,A -85,B 0,C 180,E1 21116.253,E2 21116.253} C_VEL
LIN {X 0,Y 455.248,Z 189.121,A -85,B 0,C 180,E1 21113.008,E2 21113.008} C_VEL
LIN {X 0,Y 452.012,Z 164.082,A -85,B 0,C 180,E1 21112.214,E2 21112.214} C_VEL
LIN {X 0,Y 452.081,Z 161.76,A -85,B 0,C 180,E1 21112.012,E2 21112.012} C_VEL
LIN {X 0,Y 444.774,Z 142.628,A -85,B 0,C 180,E1 21109.548,E2 21109.548} C_VEL
LIN {X 0,Y 438.04,Z 126.691,A -85,B 0,C 180,E1 21107.306,E2 21107.306} C_VEL
LIN {X 0,Y 434.393,Z 118.742,A -85,B 0,C 180,E1 21106.091,E2 21106.091} C_VEL
LIN {X 0,Y 433.22,Z 115.514,A -85,B 0,C 180,E1 21105.59,E2 21105.59} C_VEL
LIN {X 0,Y 433.234,Z 115.522,A -85,B 0,C 180,E1 21101.834,E2 21101.834} C_VEL
LIN {X 0,Y 433.246,Z 115.464,A -85,B 0,C 180,E1 21098.098,E2 21098.098} C_VEL
LIN {X 0,Y 433.246,Z 115.515,A -85,B 0,C 180,E1 21094.271,E2 21094.271} C_VEL
LIN {X 0,Y 433.235,Z 115.521,A -85,B 0,C 180,E1 21090.513,E2 21090.513} C_VEL
LIN {X 0,Y 433.209,Z 115.52,A -85,B 0,C 180,E1 21086.896,E2 21086.896} C_VEL
LIN {X 0,Y 433.199,Z 115.511,A -85,B 0,C 180,E1 21083.246,E2 21083.246} C_VEL
LIN {X 0,Y 433.2,Z 115.507,A -85,B 0,C 180,E1 21079.412,E2 21079.412} C_VEL
LIN {X 0,Y 433.204,Z 115.521,A -85,B 0,C 180,E1 21075.667,E2 21075.667} C_VEL
LIN {X 0,Y 433.232,Z 115.504,A -85,B 0,C 180,E1 21072.123,E2 21072.123} C_VEL
LIN {X 0,Y 433.247,Z 115.503,A -85,B 0,C 180,E1 21068.36,E2 21068.36} C_VEL
LIN {X 0,Y 433.239,Z 115.518,A -85,B 0,C 180,E1 21064.5,E2 21064.5} C_VEL
LIN {X 0,Y 433.229,Z 115.497,A -85,B 0,C 180,E1 21060.661,E2 21060.661} C_VEL
LIN {X 0,Y 433.208,Z 115.522,A -85,B 0,C 180,E1 21056.957,E2 21056.957} C_VEL
LIN {X 0,Y 433.194,Z 115.513,A -85,B 0,C 180,E1 21053.24,E2 21053.24} C_VEL
LIN {X 0,Y 433.19,Z 115.513,A -85,B 0,C 180,E1 21049.494,E2 21049.494} C_VEL
LIN {X 0,Y 433.191,Z 115.523,A -85,B 0,C 180,E1 21045.701,E2 21045.701} C_VEL
LIN {X 0,Y 433.2,Z 115.504,A -85,B 0,C 180,E1 21041.984,E2 21041.984} C_VEL
LIN {X 0,Y 433.223,Z 115.512,A -85,B 0,C 180,E1 21038.329,E2 21038.329} C_VEL
LIN {X 0,Y 433.234,Z 115.517,A -85,B 0,C 180,E1 21034.579,E2 21034.579} C_VEL
LIN {X 0,Y 433.24,Z 115.502,A -85,B 0,C 180,E1 21030.707,E2 21030.707} C_VEL
LIN {X 0,Y 433.221,Z 115.506,A -85,B 0,C 180,E1 21026.906,E2 21026.906} C_VEL
LIN {X 0,Y 433.198,Z 115.514,A -85,B 0,C 180,E1 21023.215,E2 21023.215} C_VEL
LIN {X 0,Y 433.185,Z 115.519,A -85,B 0,C 180,E1 21019.564,E2 21019.564} C_VEL
LIN {X 0,Y 433.183,Z 115.515,A -85,B 0,C 180,E1 21015.807,E2 21015.807} C_VEL
LIN {X 0,Y 433.186,Z 115.522,A -85,B 0,C 180,E1 21011.993,E2 21011.993} C_VEL
LIN {X 0,Y 433.208,Z 115.602,A -85,B 0,C 180,E1 21010.258,E2 21010.258} C_VEL
LIN {X 0,Y 434.536,Z 119.071,A -85,B 0,C 180,E1 21009.674,E2 21009.674} C_VEL
LIN {X 0,Y 441.486,Z 136.671,A -85,B 0,C 180,E1 21006.813,E2 21006.813} C_VEL
LIN {X 0,Y 447.981,Z 154.974,A -85,B 0,C 180,E1 21004.101,E2 21004.101} C_VEL
LIN {X 0,Y 449.225,Z 158.719,A -85,B 0,C 180,E1 21003.579,E2 21003.579} C_VEL
LIN {X 0,Y 447.991,Z 173.851,A -85,B 0,C 180,E1 21002.103,E2 21002.103} C_VEL
LIN {X 0,Y 453.074,Z 203.579,A -85,B 0,C 180,E1 21001.125,E2 21001.125} C_VEL
LIN {X 0,Y 450.78,Z 351.618,A -85,B 0,C 180,E1 20998.814,E2 20998.814} C_VEL
LIN {X 0,Y 449.832,Z 359.319,A -85,B 0,C 180,E1 20998.763,E2 20998.763} C_VEL
LIN {X 0,Y 444.172,Z 379.794,A -85,B 0,C 180,E1 20998.866,E2 20998.866} C_VEL
LIN {X 0,Y 443.428,Z 386.384,A -85,B 0,C 180,E1 20998.795,E2 20998.795} C_VEL
LIN {X 0,Y 442.703,Z 405.604,A -85,B 0,C 180,E1 20998.312,E2 20998.312} C_VEL
LIN {X 0,Y 441.597,Z 423.779,A -85,B 0,C 180,E1 20997.618,E2 20997.618} C_VEL
LIN {X 0,Y 440.165,Z 441.003,A -85,B 0,C 180,E1 20996.728,E2 20996.728} C_VEL
LIN {X 0,Y 438.31,Z 458.802,A -85,B 0,C 180,E1 20995.539,E2 20995.539} C_VEL
LIN {X 0,Y 436.292,Z 475.35,A -85,B 0,C 180,E1 20994.145,E2 20994.145} C_VEL
LIN {X 0,Y 434.234,Z 490.437,A -85,B 0,C 180,E1 20992.581,E2 20992.581} C_VEL
LIN {X 0,Y 432.201,Z 504.31,A -85,B 0,C 180,E1 20990.832,E2 20990.832} C_VEL
LIN {X 0,Y 430.227,Z 517.311,A -85,B 0,C 180,E1 20988.846,E2 20988.846} C_VEL
LIN {X 0,Y 428.46,Z 528.936,A -85,B 0,C 180,E1 20986.679,E2 20986.679} C_VEL
LIN {X 0,Y 427.009,Z 539.005,A -85,B 0,C 180,E1 20984.37,E2 20984.37} C_VEL
LIN {X 0,Y 425.923,Z 547.103,A -85,B 0,C 180,E1 20982.059,E2 20982.059} C_VEL
LIN {X 0,Y 425.14,Z 553.831,A -85,B 0,C 180,E1 20979.611,E2 20979.611} C_VEL
LIN {X 0,Y 424.64,Z 559.098,A -85,B 0,C 180,E1 20977.032,E2 20977.032} C_VEL
LIN {X 0,Y 424.37,Z 562.639,A -85,B 0,C 180,E1 20974.458,E2 20974.458} C_VEL
LIN {X 0,Y 424.252,Z 564.635,A -85,B 0,C 180,E1 20971.755,E2 20971.755} C_VEL
LIN {X 0,Y 424.234,Z 564.942,A -85,B 0,C 180,E1 20969.189,E2 20969.189} C_VEL
LIN {X 0,Y 424.305,Z 563.614,A -85,B 0,C 180,E1 20966.487,E2 20966.487} C_VEL
LIN {X 0,Y 424.51,Z 560.729,A -85,B 0,C 180,E1 20963.915,E2 20963.915} C_VEL
LIN {X 0,Y 424.913,Z 556.172,A -85,B 0,C 180,E1 20961.338,E2 20961.338} C_VEL
LIN {X 0,Y 425.602,Z 549.807,A -85,B 0,C 180,E1 20958.755,E2 20958.755} C_VEL
LIN {X 0,Y 426.614,Z 541.912,A -85,B 0,C 180,E1 20956.306,E2 20956.306} C_VEL
LIN {X 0,Y 427.938,Z 532.535,A -85,B 0,C 180,E1 20953.995,E2 20953.995} C_VEL
LIN {X 0,Y 429.563,Z 521.699,A -85,B 0,C 180,E1 20951.825,E2 20951.825} C_VEL
LIN {X 0,Y 431.449,Z 509.376,A -85,B 0,C 180,E1 20949.799,E2 20949.799} C_VEL
LIN {X 0,Y 433.447,Z 495.999,A -85,B 0,C 180,E1 20947.984,E2 20947.984} C_VEL
LIN {X 0,Y 435.501,Z 481.475,A -85,B 0,C 180,E1 20946.357,E2 20946.357} C_VEL
LIN {X 0,Y 437.514,Z 465.783,A -85,B 0,C 180,E1 20944.916,E2 20944.916} C_VEL
LIN {X 0,Y 439.308,Z 449.885,A -85,B 0,C 180,E1 20943.733,E2 20943.733} C_VEL
LIN {X 0,Y 440.893,Z 433.037,A -85,B 0,C 180,E1 20942.735,E2 20942.735} C_VEL
LIN {X 0,Y 442.247,Z 414.359,A -85,B 0,C 180,E1 20941.898,E2 20941.898} C_VEL
LIN {X 0,Y 443.18,Z 395.015,A -85,B 0,C 180,E1 20941.296,E2 20941.296} C_VEL
LIN {X 0,Y 443.738,Z 369.713,A -85,B 0,C 180,E1 20940.833,E2 20940.833} C_VEL
LIN {X 0,Y 446.363,Z 203.072,A -85,B 0,C 180,E1 20938.181,E2 20938.181} C_VEL
LIN {X 0,Y 441.125,Z 172.964,A -85,B 0,C 180,E1 20937.121,E2 20937.121} C_VEL
LIN {X 0,Y 442.091,Z 161.549,A -85,B 0,C 180,E1 20935.96,E2 20935.96} C_VEL
LIN {X 0,Y 435.911,Z 143.506,A -85,B 0,C 180,E1 20933.289,E2 20933.289} C_VEL
LIN {X 0,Y 429.294,Z 126.551,A -85,B 0,C 180,E1 20930.517,E2 20930.517} C_VEL
LIN {X 0,Y 426.264,Z 119.382,A -85,B 0,C 180,E1 20929.257,E2 20929.257} C_VEL
LIN {X 0,Y 425.292,Z 116.503,A -85,B 0,C 180,E1 20928.741,E2 20928.741} C_VEL
LIN {X 0,Y 425.306,Z 116.51,A -85,B 0,C 180,E1 20924.957,E2 20924.957} C_VEL
LIN {X 0,Y 425.32,Z 116.505,A -85,B 0,C 180,E1 20921.166,E2 20921.166} C_VEL
LIN {X 0,Y 425.33,Z 116.589,A -85,B 0,C 180,E1 20918.263,E2 20918.263} C_VEL
LIN {X 0,Y 435.024,Z 143.291,A -85,B 0,C 180,E1 20914.976,E2 20914.976} C_VEL
LIN {X 0,Y 439.158,Z 155.977,A -85,B 0,C 180,E1 20913.485,E2 20913.485} C_VEL
LIN {X 0,Y 438.028,Z 184.054,A -85,B 0,C 180,E1 20911.06,E2 20911.06} C_VEL
LIN {X 0,Y 440.576,Z 202.401,A -85,B 0,C 180,E1 20910.479,E2 20910.479} C_VEL
LIN {X 0,Y 435.499,Z 395.062,A -85,B 0,C 180,E1 20906.698,E2 20906.698} C_VEL
LIN {X 0,Y 434.778,Z 414.709,A -85,B 0,C 180,E1 20906.056,E2 20906.056} C_VEL
LIN {X 0,Y 433.873,Z 432.647,A -85,B 0,C 180,E1 20905.235,E2 20905.235} C_VEL
LIN {X 0,Y 432.788,Z 449.94,A -85,B 0,C 180,E1 20904.21,E2 20904.21} C_VEL
LIN {X 0,Y 431.591,Z 466.577,A -85,B 0,C 180,E1 20902.975,E2 20902.975} C_VEL
LIN {X 0,Y 430.331,Z 482.387,A -85,B 0,C 180,E1 20901.538,E2 20901.538} C_VEL
LIN {X 0,Y 429.056,Z 497.332,A -85,B 0,C 180,E1 20899.891,E2 20899.891} C_VEL
LIN {X 0,Y 427.883,Z 510.789,A -85,B 0,C 180,E1 20898.107,E2 20898.107} C_VEL
LIN {X 0,Y 426.839,Z 522.927,A -85,B 0,C 180,E1 20896.173,E2 20896.173} C_VEL
LIN {X 0,Y 425.981,Z 533.556,A -85,B 0,C 180,E1 20894.129,E2 20894.129} C_VEL
LIN {X 0,Y 425.294,Z 542.871,A -85,B 0,C 180,E1 20891.94,E2 20891.94} C_VEL
LIN {X 0,Y 424.801,Z 550.74,A -85,B 0,C 180,E1 20889.62,E2 20889.62} C_VEL
LIN {X 0,Y 424.497,Z 556.766,A -85,B 0,C 180,E1 20887.308,E2 20887.308} C_VEL
LIN {X 0,Y 424.323,Z 561.342,A -85,B 0,C 180,E1 20884.866,E2 20884.866} C_VEL
LIN {X 0,Y 424.26,Z 564.168,A -85,B 0,C 180,E1 20882.432,E2 20882.432} C_VEL
LIN {X 0,Y 424.259,Z 565.319,A -85,B 0,C 180,E1 20880,E2 20880} C_VEL
LIN {X 0,Y 424.303,Z 564.804,A -85,B 0,C 180,E1 20877.569,E2 20877.569} C_VEL
LIN {X 0,Y 424.425,Z 562.613,A -85,B 0,C 180,E1 20875.135,E2 20875.135} C_VEL
LIN {X 0,Y 424.662,Z 558.691,A -85,B 0,C 180,E1 20872.696,E2 20872.696} C_VEL
LIN {X 0,Y 425.057,Z 552.884,A -85,B 0,C 180,E1 20870.249,E2 20870.249} C_VEL
LIN {X 0,Y 425.642,Z 545.514,A -85,B 0,C 180,E1 20867.933,E2 20867.933} C_VEL
LIN {X 0,Y 426.427,Z 536.698,A -85,B 0,C 180,E1 20865.748,E2 20865.748} C_VEL
LIN {X 0,Y 427.384,Z 526.471,A -85,B 0,C 180,E1 20863.696,E2 20863.696} C_VEL
LIN {X 0,Y 428.517,Z 514.565,A -85,B 0,C 180,E1 20861.743,E2 20861.743} C_VEL
LIN {X 0,Y 429.779,Z 501.232,A -85,B 0,C 180,E1 20859.931,E2 20859.931} C_VEL
LIN {X 0,Y 431.09,Z 486.476,A -85,B 0,C 180,E1 20858.285,E2 20858.285} C_VEL
LIN {X 0,Y 432.434,Z 470.065,A -85,B 0,C 180,E1 20856.783,E2 20856.783} C_VEL
LIN {X 0,Y 433.632,Z 453.332,A -85,B 0,C 180,E1 20855.551,E2 20855.551} C_VEL
LIN {X 0,Y 434.705,Z 435.023,A -85,B 0,C 180,E1 20854.489,E2 20854.489} C_VEL
LIN {X 0,Y 435.586,Z 415.744,A -85,B 0,C 180,E1 20853.639,E2 20853.639} C_VEL
LIN {X 0,Y 436.221,Z 396.077,A -85,B 0,C 180,E1 20853.033,E2 20853.033} C_VEL
LIN {X 0,Y 439.42,Z 309.939,A -85,B 0,C 180,E1 20851.099,E2 20851.099} C_VEL
LIN {X 0,Y 444.479,Z 220.14,A -85,B 0,C 180,E1 20848.89,E2 20848.89} C_VEL
LIN {X 0,Y 445.492,Z 202.346,A -85,B 0,C 180,E1 20848.415,E2 20848.415} C_VEL
LIN {X 0,Y 444.713,Z 195.339,A -85,B 0,C 180,E1 20848.03,E2 20848.03} C_VEL
LIN {X 0,Y 446.661,Z 160.413,A -85,B 0,C 180,E1 20845.016,E2 20845.016} C_VEL
LIN {X 0,Y 443.752,Z 150.549,A -85,B 0,C 180,E1 20843.552,E2 20843.552} C_VEL
LIN {X 0,Y 440.071,Z 141.342,A -85,B 0,C 180,E1 20841.826,E2 20841.826} C_VEL
LIN {X 0,Y 437.811,Z 136.785,A -85,B 0,C 180,E1 20840.733,E2 20840.733} C_VEL
LIN {X 0,Y 436.094,Z 133.277,A -85,B 0,C 180,E1 20839.774,E2 20839.774} C_VEL
LIN {X 0,Y 434.019,Z 129.488,A -85,B 0,C 180,E1 20838.48,E2 20838.48} C_VEL
LIN {X 0,Y 433.627,Z 128.575,A -85,B 0,C 180,E1 20838.141,E2 20838.141} C_VEL
LIN {X 0,Y 431.287,Z 125.979,A -85,B 0,C 180,E1 20836.118,E2 20836.118} C_VEL
LIN {X 0,Y 430.844,Z 124.57,A -85,B 0,C 180,E1 20834.496,E2 20834.496} C_VEL
LIN {X 0,Y 430.02,Z 127.507,A -85,B 0,C 180,E1 20833.543,E2 20833.543} C_VEL
LIN {X 0,Y 437.548,Z 144.932,A -85,B 0,C 180,E1 20830.984,E2 20830.984} C_VEL
LIN {X 0,Y 445.123,Z 164.753,A -85,B 0,C 180,E1 20828.377,E2 20828.377} C_VEL
LIN {X 0,Y 448.702,Z 192.32,A -85,B 0,C 180,E1 20827.498,E2 20827.498} C_VEL
LIN {X 0,Y 443.003,Z 412.96,A -85,B 0,C 180,E1 20823.516,E2 20823.516} C_VEL
LIN {X 0,Y 442,Z 433.879,A -85,B 0,C 180,E1 20822.999,E2 20822.999} C_VEL
LIN {X 0,Y 440.634,Z 453.657,A -85,B 0,C 180,E1 20822.293,E2 20822.293} C_VEL
LIN {X 0,Y 438.889,Z 474.366,A -85,B 0,C 180,E1 20821.294,E2 20821.294} C_VEL
LIN {X 0,Y 436.944,Z 494.091,A -85,B 0,C 180,E1 20820.076,E2 20820.076} C_VEL
LIN {X 0,Y 434.904,Z 512.89,A -85,B 0,C 180,E1 20818.644,E2 20818.644} C_VEL
LIN {X 0,Y 432.965,Z 530.104,A -85,B 0,C 180,E1 20817.062,E2 20817.062} C_VEL
LIN {X 0,Y 430.976,Z 547.11,A -85,B 0,C 180,E1 20815.205,E2 20815.205} C_VEL
LIN {X 0,Y 429.147,Z 563.194,A -85,B 0,C 180,E1 20813.116,E2 20813.116} C_VEL
LIN {X 0,Y 427.624,Z 577.228,A -85,B 0,C 180,E1 20810.962,E2 20810.962} C_VEL
LIN {X 0,Y 426.373,Z 589.906,A -85,B 0,C 180,E1 20808.668,E2 20808.668} C_VEL
LIN {X 0,Y 425.362,Z 601.73,A -85,B 0,C 180,E1 20806.104,E2 20806.104} C_VEL
LIN {X 0,Y 424.669,Z 611.618,A -85,B 0,C 180,E1 20803.48,E2 20803.48} C_VEL
LIN {X 0,Y 424.297,Z 619.088,A -85,B 0,C 180,E1 20801.005,E2 20801.005} C_VEL
LIN {X 0,Y 424.097,Z 625.207,A -85,B 0,C 180,E1 20798.406,E2 20798.406} C_VEL
LIN {X 0,Y 424.028,Z 629.642,A -85,B 0,C 180,E1 20795.82,E2 20795.82} C_VEL
LIN {X 0,Y 424.024,Z 632.417,A -85,B 0,C 180,E1 20793.245,E2 20793.245} C_VEL
LIN {X 0,Y 424.034,Z 633.574,A -85,B 0,C 180,E1 20790.676,E2 20790.676} C_VEL
LIN {X 0,Y 424.029,Z 633.151,A -85,B 0,C 180,E1 20787.974,E2 20787.974} C_VEL
LIN {X 0,Y 424.017,Z 631.182,A -85,B 0,C 180,E1 20785.402,E2 20785.402} C_VEL
LIN {X 0,Y 424.055,Z 627.528,A -85,B 0,C 180,E1 20782.822,E2 20782.822} C_VEL
LIN {X 0,Y 424.184,Z 622.221,A -85,B 0,C 180,E1 20780.23,E2 20780.23} C_VEL
LIN {X 0,Y 424.472,Z 615.145,A -85,B 0,C 180,E1 20777.623,E2 20777.623} C_VEL
LIN {X 0,Y 424.995,Z 606.685,A -85,B 0,C 180,E1 20775.142,E2 20775.142} C_VEL
LIN {X 0,Y 425.801,Z 596.26,A -85,B 0,C 180,E1 20772.65,E2 20772.65} C_VEL
LIN {X 0,Y 426.901,Z 584.397,A -85,B 0,C 180,E1 20770.291,E2 20770.291} C_VEL
LIN {X 0,Y 428.263,Z 571.174,A -85,B 0,C 180,E1 20768.066,E2 20768.066} C_VEL
LIN {X 0,Y 429.949,Z 556.061,A -85,B 0,C 180,E1 20765.914,E2 20765.914} C_VEL
LIN {X 0,Y 431.888,Z 539.326,A -85,B 0,C 180,E1 20763.906,E2 20763.906} C_VEL
LIN {X 0,Y 433.861,Z 522.248,A -85,B 0,C 180,E1 20762.183,E2 20762.183} C_VEL
LIN {X 0,Y 435.87,Z 504.148,A -85,B 0,C 180,E1 20760.656,E2 20760.656} C_VEL
LIN {X 0,Y 437.89,Z 484.768,A -85,B 0,C 180,E1 20759.315,E2 20759.315} C_VEL
LIN {X 0,Y 439.797,Z 463.888,A -85,B 0,C 180,E1 20758.168,E2 20758.168} C_VEL
LIN {X 0,Y 441.434,Z 442.873,A -85,B 0,C 180,E1 20757.295,E2 20757.295} C_VEL
LIN {X 0,Y 442.688,Z 421.214,A -85,B 0,C 180,E1 20756.66,E2 20756.66} C_VEL
LIN {X 0,Y 444.954,Z 335.584,A -85,B 0,C 180,E1 20755.079,E2 20755.079} C_VEL
LIN {X 0,Y 448.561,Z 189.99,A -85,B 0,C 180,E1 20752.445,E2 20752.445} C_VEL
LIN {X 0,Y 445.104,Z 164.735,A -85,B 0,C 180,E1 20751.626,E2 20751.626} C_VEL
LIN {X 0,Y 437.972,Z 146.095,A -85,B 0,C 180,E1 20749.182,E2 20749.182} C_VEL
LIN {X 0,Y 430.246,Z 127.915,A -85,B 0,C 180,E1 20746.539,E2 20746.539} C_VEL
LIN {X 0,Y 426.512,Z 119.9,A -85,B 0,C 180,E1 20745.26,E2 20745.26} C_VEL
LIN {X 0,Y 425.278,Z 116.512,A -85,B 0,C 180,E1 20744.718,E2 20744.718} C_VEL
LIN {X 0,Y 425.265,Z 116.501,A -85,B 0,C 180,E1 20740.993,E2 20740.993} C_VEL
LIN {X 0,Y 425.26,Z 116.47,A -85,B 0,C 180,E1 20737.153,E2 20737.153} C_VEL
LIN {X 0,Y 425.265,Z 116.497,A -85,B 0,C 180,E1 20733.378,E2 20733.378} C_VEL
LIN {X 0,Y 425.272,Z 116.501,A -85,B 0,C 180,E1 20729.586,E2 20729.586} C_VEL
LIN {X 0,Y 425.291,Z 116.508,A -85,B 0,C 180,E1 20725.931,E2 20725.931} C_VEL
LIN {X 0,Y 425.304,Z 116.505,A -85,B 0,C 180,E1 20722.095,E2 20722.095} C_VEL
LIN {X 0,Y 425.303,Z 116.488,A -85,B 0,C 180,E1 20718.22,E2 20718.22} C_VEL
LIN {X 0,Y 425.309,Z 116.493,A -85,B 0,C 180,E1 20714.408,E2 20714.408} C_VEL
LIN {X 0,Y 425.294,Z 116.507,A -85,B 0,C 180,E1 20710.566,E2 20710.566} C_VEL
LIN {X 0,Y 425.269,Z 116.486,A -85,B 0,C 180,E1 20706.886,E2 20706.886} C_VEL
LIN {X 0,Y 425.259,Z 116.51,A -85,B 0,C 180,E1 20703.235,E2 20703.235} C_VEL
LIN {X 0,Y 425.254,Z 116.505,A -85,B 0,C 180,E1 20699.461,E2 20699.461} C_VEL
LIN {X 0,Y 425.254,Z 116.498,A -85,B 0,C 180,E1 20695.685,E2 20695.685} C_VEL
LIN {X 0,Y 425.271,Z 116.512,A -85,B 0,C 180,E1 20692.026,E2 20692.026} C_VEL
LIN {X 0,Y 425.289,Z 116.486,A -85,B 0,C 180,E1 20688.335,E2 20688.335} C_VEL
LIN {X 0,Y 425.304,Z 116.505,A -85,B 0,C 180,E1 20684.549,E2 20684.549} C_VEL
LIN {X 0,Y 425.296,Z 116.5,A -85,B 0,C 180,E1 20680.641,E2 20680.641} C_VEL
LIN {X 0,Y 425.285,Z 116.489,A -85,B 0,C 180,E1 20676.814,E2 20676.814} C_VEL
LIN {X 0,Y 425.274,Z 116.503,A -85,B 0,C 180,E1 20673.005,E2 20673.005} C_VEL
LIN {X 0,Y 425.254,Z 116.511,A -85,B 0,C 180,E1 20669.322,E2 20669.322} C_VEL
LIN {X 0,Y 425.247,Z 116.51,A -85,B 0,C 180,E1 20665.615,E2 20665.615} C_VEL
LIN {X 0,Y 425.246,Z 116.508,A -85,B 0,C 180,E1 20661.748,E2 20661.748} C_VEL
LIN {X 0,Y 425.247,Z 116.512,A -85,B 0,C 180,E1 20657.925,E2 20657.925} C_VEL
LIN {X 0,Y 425.253,Z 116.515,A -85,B 0,C 180,E1 20654.102,E2 20654.102} C_VEL
LIN {X 0,Y 425.292,Z 116.646,A -85,B 0,C 180,E1 20651.106,E2 20651.106} C_VEL
LIN {X 0,Y 432.774,Z 135.294,A -85,B 0,C 180,E1 20647.918,E2 20647.918} C_VEL
LIN {X 0,Y 439.275,Z 153.073,A -85,B 0,C 180,E1 20645.159,E2 20645.159} C_VEL
LIN {X 0,Y 442.157,Z 161.763,A -85,B 0,C 180,E1 20643.91,E2 20643.91} C_VEL
LIN {X 0,Y 441.145,Z 173.819,A -85,B 0,C 180,E1 20642.729,E2 20642.729} C_VEL
LIN {X 0,Y 446.433,Z 204.797,A -85,B 0,C 180,E1 20641.681,E2 20641.681} C_VEL
LIN {X 0,Y 443.428,Z 386.384,A -85,B 0,C 180,E1 20638.795,E2 20638.795} C_VEL
LIN {X 0,Y 442.14,Z 395.136,A -85,B 0,C 180,E1 20638.694,E2 20638.694} C_VEL
LIN {X 0,Y 436.655,Z 412.138,A -85,B 0,C 180,E1 20638.561,E2 20638.561} C_VEL
LIN {X 0,Y 435.059,Z 419.556,A -85,B 0,C 180,E1 20638.351,E2 20638.351} C_VEL
LIN {X 0,Y 434.954,Z 420.592,A -85,B 0,C 180,E1 20638.307,E2 20638.307} C_VEL
LIN {X 0,Y 433.56,Z 437.663,A -85,B 0,C 180,E1 20637.466,E2 20637.466} C_VEL
LIN {X 0,Y 431.807,Z 454.464,A -85,B 0,C 180,E1 20636.395,E2 20636.395} C_VEL
LIN {X 0,Y 429.75,Z 471.223,A -85,B 0,C 180,E1 20635.051,E2 20635.051} C_VEL
LIN {X 0,Y 427.556,Z 486.873,A -85,B 0,C 180,E1 20633.497,E2 20633.497} C_VEL
LIN {X 0,Y 425.331,Z 501.424,A -85,B 0,C 180,E1 20631.73,E2 20631.73} C_VEL
LIN {X 0,Y 423.195,Z 514.828,A -85,B 0,C 180,E1 20629.745,E2 20629.745} C_VEL
LIN {X 0,Y 421.333,Z 526.329,A -85,B 0,C 180,E1 20627.682,E2 20627.682} C_VEL
LIN {X 0,Y 419.654,Z 537,A -85,B 0,C 180,E1 20625.334,E2 20625.334} C_VEL
LIN {X 0,Y 418.389,Z 545.635,A -85,B 0,C 180,E1 20622.981,E2 20622.981} C_VEL
LIN {X 0,Y 417.407,Z 553.182,A -85,B 0,C 180,E1 20620.349,E2 20620.349} C_VEL
LIN {X 0,Y 416.795,Z 558.815,A -85,B 0,C 180,E1 20617.72,E2 20617.72} C_VEL
LIN {X 0,Y 416.455,Z 562.703,A -85,B 0,C 180,E1 20615.096,E2 20615.096} C_VEL
LIN {X 0,Y 416.299,Z 564.97,A -85,B 0,C 180,E1 20612.477,E2 20612.477} C_VEL
LIN {X 0,Y 416.261,Z 565.67,A -85,B 0,C 180,E1 20609.724,E2 20609.724} C_VEL
LIN {X 0,Y 416.309,Z 564.784,A -85,B 0,C 180,E1 20607.108,E2 20607.108} C_VEL
LIN {X 0,Y 416.487,Z 562.339,A -85,B 0,C 180,E1 20604.489,E2 20604.489} C_VEL
LIN {X 0,Y 416.859,Z 558.245,A -85,B 0,C 180,E1 20601.864,E2 20601.864} C_VEL
LIN {X 0,Y 417.506,Z 552.376,A -85,B 0,C 180,E1 20599.233,E2 20599.233} C_VEL
LIN {X 0,Y 418.479,Z 545.024,A -85,B 0,C 180,E1 20596.739,E2 20596.739} C_VEL
LIN {X 0,Y 419.778,Z 536.251,A -85,B 0,C 180,E1 20594.385,E2 20594.385} C_VEL
LIN {X 0,Y 421.492,Z 525.362,A -85,B 0,C 180,E1 20592.037,E2 20592.037} C_VEL
LIN {X 0,Y 423.391,Z 513.685,A -85,B 0,C 180,E1 20589.975,E2 20589.975} C_VEL
LIN {X 0,Y 425.481,Z 500.545,A -85,B 0,C 180,E1 20588.059,E2 20588.059} C_VEL
LIN {X 0,Y 427.72,Z 485.789,A -85,B 0,C 180,E1 20586.291,E2 20586.291} C_VEL
LIN {X 0,Y 429.926,Z 469.963,A -85,B 0,C 180,E1 20584.745,E2 20584.745} C_VEL
LIN {X 0,Y 431.903,Z 453.771,A -85,B 0,C 180,E1 20583.461,E2 20583.461} C_VEL
LIN {X 0,Y 433.665,Z 436.808,A -85,B 0,C 180,E1 20582.391,E2 20582.391} C_VEL
LIN {X 0,Y 435.15,Z 418.289,A -85,B 0,C 180,E1 20581.501,E2 20581.501} C_VEL
LIN {X 0,Y 436.208,Z 399.509,A -85,B 0,C 180,E1 20580.859,E2 20580.859} C_VEL
LIN {X 0,Y 436.799,Z 379.623,A -85,B 0,C 180,E1 20580.436,E2 20580.436} C_VEL
LIN {X 0,Y 439.777,Z 204.476,A -85,B 0,C 180,E1 20577.611,E2 20577.611} C_VEL
LIN {X 0,Y 434.341,Z 172.77,A -85,B 0,C 180,E1 20576.462,E2 20576.462} C_VEL
LIN {X 0,Y 435.02,Z 164.503,A -85,B 0,C 180,E1 20575.603,E2 20575.603} C_VEL
LIN {X 0,Y 428.747,Z 146.275,A -85,B 0,C 180,E1 20572.842,E2 20572.842} C_VEL
LIN {X 0,Y 422.517,Z 130.28,A -85,B 0,C 180,E1 20570.167,E2 20570.167} C_VEL
LIN {X 0,Y 418.41,Z 120.593,A -85,B 0,C 180,E1 20568.415,E2 20568.415} C_VEL
LIN {X 0,Y 417.374,Z 117.498,A -85,B 0,C 180,E1 20567.873,E2 20567.873} C_VEL
LIN {X 0,Y 417.375,Z 117.485,A -85,B 0,C 180,E1 20564.005,E2 20564.005} C_VEL
LIN {X 0,Y 417.382,Z 117.496,A -85,B 0,C 180,E1 20560.121,E2 20560.121} C_VEL
LIN {X 0,Y 417.387,Z 117.591,A -85,B 0,C 180,E1 20558.872,E2 20558.872} C_VEL
LIN {X 0,Y 426.86,Z 143.378,A -85,B 0,C 180,E1 20555.629,E2 20555.629} C_VEL
LIN {X 0,Y 431.933,Z 158.82,A -85,B 0,C 180,E1 20553.794,E2 20553.794} C_VEL
LIN {X 0,Y 430.846,Z 184.544,A -85,B 0,C 180,E1 20551.555,E2 20551.555} C_VEL
LIN {X 0,Y 433.448,Z 203.618,A -85,B 0,C 180,E1 20550.943,E2 20550.943} C_VEL
LIN {X 0,Y 428.044,Z 395.783,A -85,B 0,C 180,E1 20547.074,E2 20547.074} C_VEL
LIN {X 0,Y 427.277,Z 415.501,A -85,B 0,C 180,E1 20546.413,E2 20546.413} C_VEL
LIN {X 0,Y 426.318,Z 433.606,A -85,B 0,C 180,E1 20545.566,E2 20545.566} C_VEL
LIN {X 0,Y 425.114,Z 451.829,A -85,B 0,C 180,E1 20544.453,E2 20544.453} C_VEL
LIN {X 0,Y 423.809,Z 469.046,A -85,B 0,C 180,E1 20543.13,E2 20543.13} C_VEL
LIN {X 0,Y 422.449,Z 485.273,A -85,B 0,C 180,E1 20541.595,E2 20541.595} C_VEL
LIN {X 0,Y 421.152,Z 499.856,A -85,B 0,C 180,E1 20539.923,E2 20539.923} C_VEL
LIN {X 0,Y 419.909,Z 513.543,A -85,B 0,C 180,E1 20538.032,E2 20538.032} C_VEL
LIN {X 0,Y 418.792,Z 526.063,A -85,B 0,C 180,E1 20535.936,E2 20535.936} C_VEL
LIN {X 0,Y 417.877,Z 536.93,A -85,B 0,C 180,E1 20533.703,E2 20533.703} C_VEL
LIN {X 0,Y 417.206,Z 545.914,A -85,B 0,C 180,E1 20531.42,E2 20531.42} C_VEL
LIN {X 0,Y 416.755,Z 553.12,A -85,B 0,C 180,E1 20529.111,E2 20529.111} C_VEL
LIN {X 0,Y 416.482,Z 558.724,A -85,B 0,C 180,E1 20526.756,E2 20526.756} C_VEL
LIN {X 0,Y 416.326,Z 562.864,A -85,B 0,C 180,E1 20524.27,E2 20524.27} C_VEL
LIN {X 0,Y 416.275,Z 565.271,A -85,B 0,C 180,E1 20521.79,E2 20521.79} C_VEL
LIN {X 0,Y 416.298,Z 566.004,A -85,B 0,C 180,E1 20519.312,E2 20519.312} C_VEL
LIN {X 0,Y 416.363,Z 565.066,A -85,B 0,C 180,E1 20516.834,E2 20516.834} C_VEL
LIN {X 0,Y 416.527,Z 562.432,A -85,B 0,C 180,E1 20514.352,E2 20514.352} C_VEL
LIN {X 0,Y 416.84,Z 558.02,A -85,B 0,C 180,E1 20511.864,E2 20511.864} C_VEL
LIN {X 0,Y 417.304,Z 552.11,A -85,B 0,C 180,E1 20509.508,E2 20509.508} C_VEL
LIN {X 0,Y 418.009,Z 544.329,A -85,B 0,C 180,E1 20507.147,E2 20507.147} C_VEL
LIN {X 0,Y 418.919,Z 535.008,A -85,B 0,C 180,E1 20504.921,E2 20504.921} C_VEL
LIN {X 0,Y 420.029,Z 524.242,A -85,B 0,C 180,E1 20502.832,E2 20502.832} C_VEL
LIN {X 0,Y 421.34,Z 511.51,A -85,B 0,C 180,E1 20500.818,E2 20500.818} C_VEL
LIN {X 0,Y 422.732,Z 497.49,A -85,B 0,C 180,E1 20499.002,E2 20499.002} C_VEL
LIN {X 0,Y 424.136,Z 482.514,A -85,B 0,C 180,E1 20497.403,E2 20497.403} C_VEL
LIN {X 0,Y 425.532,Z 465.797,A -85,B 0,C 180,E1 20495.949,E2 20495.949} C_VEL
LIN {X 0,Y 426.828,Z 448.242,A -85,B 0,C 180,E1 20494.719,E2 20494.719} C_VEL
LIN {X 0,Y 427.907,Z 430.1,A -85,B 0,C 180,E1 20493.726,E2 20493.726} C_VEL
LIN {X 0,Y 428.806,Z 410.228,A -85,B 0,C 180,E1 20492.92,E2 20492.92} C_VEL
LIN {X 0,Y 429.492,Z 388.342,A -85,B 0,C 180,E1 20492.322,E2 20492.322} C_VEL
LIN {X 0,Y 432.904,Z 310.106,A -85,B 0,C 180,E1 20490.488,E2 20490.488} C_VEL
LIN {X 0,Y 438.457,Z 222.056,A -85,B 0,C 180,E1 20488.232,E2 20488.232} C_VEL
LIN {X 0,Y 439.637,Z 204.043,A -85,B 0,C 180,E1 20487.733,E2 20487.733} C_VEL
LIN {X 0,Y 438.884,Z 196.867,A -85,B 0,C 180,E1 20487.321,E2 20487.321} C_VEL
LIN {X 0,Y 441.063,Z 164.462,A -85,B 0,C 180,E1 20484.473,E2 20484.473} C_VEL
LIN {X 0,Y 438.36,Z 154.913,A -85,B 0,C 180,E1 20482.971,E2 20482.971} C_VEL
LIN {X 0,Y 435.663,Z 147.554,A -85,B 0,C 180,E1 20481.501,E2 20481.501} C_VEL
LIN {X 0,Y 433.299,Z 142.474,A -85,B 0,C 180,E1 20480.213,E2 20480.213} C_VEL
LIN {X 0,Y 432.086,Z 139.869,A -85,B 0,C 180,E1 20479.441,E2 20479.441} C_VEL
LIN {X 0,Y 430.434,Z 135.939,A -85,B 0,C 180,E1 20478.067,E2 20478.067} C_VEL
LIN {X 0,Y 428.311,Z 133.267,A -85,B 0,C 180,E1 20475.921,E2 20475.921} C_VEL
LIN {X 0,Y 428.11,Z 132.284,A -85,B 0,C 180,E1 20474.668,E2 20474.668} C_VEL
LIN {X 0,Y 427.249,Z 135.021,A -85,B 0,C 180,E1 20473.846,E2 20473.846} C_VEL
LIN {X 0,Y 426.712,Z 138.75,A -85,B 0,C 180,E1 20472.783,E2 20472.783} C_VEL
LIN {X 0,Y 434.43,Z 157.712,A -85,B 0,C 180,E1 20470.07,E2 20470.07} C_VEL
LIN {X 0,Y 437.275,Z 165.245,A -85,B 0,C 180,E1 20469.104,E2 20469.104} C_VEL
LIN {X 0,Y 439.197,Z 169.277,A -85,B 0,C 180,E1 20468.837,E2 20468.837} C_VEL
LIN {X 0,Y 442.091,Z 193.804,A -85,B 0,C 180,E1 20468.062,E2 20468.062} C_VEL
LIN {X 0,Y 436.129,Z 412.771,A -85,B 0,C 180,E1 20464.054,E2 20464.054} C_VEL
LIN {X 0,Y 435.077,Z 433.673,A -85,B 0,C 180,E1 20463.528,E2 20463.528} C_VEL
LIN {X 0,Y 433.562,Z 454.223,A -85,B 0,C 180,E1 20462.778,E2 20462.778} C_VEL
LIN {X 0,Y 431.739,Z 474.704,A -85,B 0,C 180,E1 20461.768,E2 20461.768} C_VEL
LIN {X 0,Y 429.625,Z 494.945,A -85,B 0,C 180,E1 20460.488,E2 20460.488} C_VEL
LIN {X 0,Y 427.379,Z 514.405,A -85,B 0,C 180,E1 20458.958,E2 20458.958} C_VEL
LIN {X 0,Y 425.202,Z 532.503,A -85,B 0,C 180,E1 20457.226,E2 20457.226} C_VEL
LIN {X 0,Y 423.125,Z 549.133,A -85,B 0,C 180,E1 20455.323,E2 20455.323} C_VEL
LIN {X 0,Y 421.314,Z 564.058,A -85,B 0,C 180,E1 20453.304,E2 20453.304} C_VEL
LIN {X 0,Y 419.706,Z 577.995,A -85,B 0,C 180,E1 20451.084,E2 20451.084} C_VEL
LIN {X 0,Y 418.374,Z 590.753,A -85,B 0,C 180,E1 20448.678,E2 20448.678} C_VEL
LIN {X 0,Y 417.414,Z 601.474,A -85,B 0,C 180,E1 20446.276,E2 20446.276} C_VEL
LIN {X 0,Y 416.691,Z 611.298,A -85,B 0,C 180,E1 20443.601,E2 20443.601} C_VEL
LIN {X 0,Y 416.292,Z 619.074,A -85,B 0,C 180,E1 20440.939,E2 20440.939} C_VEL
LIN {X 0,Y 416.105,Z 625.033,A -85,B 0,C 180,E1 20438.29,E2 20438.29} C_VEL
LIN {X 0,Y 416.046,Z 629.307,A -85,B 0,C 180,E1 20435.656,E2 20435.656} C_VEL
LIN {X 0,Y 416.049,Z 631.981,A -85,B 0,C 180,E1 20433.032,E2 20433.032} C_VEL
LIN {X 0,Y 416.059,Z 632.977,A -85,B 0,C 180,E1 20430.414,E2 20430.414} C_VEL
LIN {X 0,Y 416.051,Z 632.425,A -85,B 0,C 180,E1 20427.797,E2 20427.797} C_VEL
LIN {X 0,Y 416.041,Z 630.339,A -85,B 0,C 180,E1 20425.176,E2 20425.176} C_VEL
LIN {X 0,Y 416.07,Z 626.598,A -85,B 0,C 180,E1 20422.545,E2 20422.545} C_VEL
LIN {X 0,Y 416.212,Z 621.141,A -85,B 0,C 180,E1 20419.901,E2 20419.901} C_VEL
LIN {X 0,Y 416.536,Z 613.919,A -85,B 0,C 180,E1 20417.243,E2 20417.243} C_VEL
LIN {X 0,Y 417.11,Z 605.322,A -85,B 0,C 180,E1 20414.712,E2 20414.712} C_VEL
LIN {X 0,Y 417.995,Z 594.806,A -85,B 0,C 180,E1 20412.172,E2 20412.172} C_VEL
LIN {X 0,Y 419.275,Z 582.058,A -85,B 0,C 180,E1 20409.626,E2 20409.626} C_VEL
LIN {X 0,Y 420.908,Z 567.62,A -85,B 0,C 180,E1 20407.221,E2 20407.221} C_VEL
LIN {X 0,Y 422.777,Z 552.049,A -85,B 0,C 180,E1 20405.044,E2 20405.044} C_VEL
LIN {X 0,Y 424.772,Z 535.819,A -85,B 0,C 180,E1 20403.133,E2 20403.133} C_VEL
LIN {X 0,Y 426.815,Z 518.921,A -85,B 0,C 180,E1 20401.453,E2 20401.453} C_VEL
LIN {X 0,Y 428.985,Z 500.493,A -85,B 0,C 180,E1 20399.928,E2 20399.928} C_VEL
LIN {X 0,Y 431.078,Z 480.864,A -85,B 0,C 180,E1 20398.6,E2 20398.6} C_VEL
LIN {X 0,Y 432.924,Z 461.639,A -85,B 0,C 180,E1 20397.563,E2 20397.563} C_VEL
LIN {X 0,Y 434.553,Z 441.364,A -85,B 0,C 180,E1 20396.724,E2 20396.724} C_VEL
LIN {X 0,Y 435.863,Z 419.767,A -85,B 0,C 180,E1 20396.095,E2 20396.095} C_VEL
LIN {X 0,Y 441.415,Z 217.365,A -85,B 0,C 180,E1 20392.364,E2 20392.364} C_VEL
LIN {X 0,Y 441.945,Z 191.042,A -85,B 0,C 180,E1 20391.871,E2 20391.871} C_VEL
LIN {X 0,Y 438.834,Z 168.165,A -85,B 0,C 180,E1 20391.111,E2 20391.111} C_VEL
LIN {X 0,Y 436.872,Z 164.372,A -85,B 0,C 180,E1 20390.828,E2 20390.828} C_VEL
LIN {X 0,Y 429.729,Z 145.901,A -85,B 0,C 180,E1 20388.285,E2 20388.285} C_VEL
LIN {X 0,Y 422.236,Z 128.629,A -85,B 0,C 180,E1 20385.654,E2 20385.654} C_VEL
LIN {X 0,Y 417.398,Z 117.76,A -85,B 0,C 180,E1 20383.862,E2 20383.862} C_VEL
LIN {X 0,Y 417.334,Z 117.489,A -85,B 0,C 180,E1 20383.44,E2 20383.44} C_VEL
LIN {X 0,Y 417.342,Z 117.45,A -85,B 0,C 180,E1 20379.734,E2 20379.734} C_VEL
LIN {X 0,Y 417.355,Z 117.484,A -85,B 0,C 180,E1 20375.931,E2 20375.931} C_VEL
LIN {X 0,Y 417.37,Z 117.483,A -85,B 0,C 180,E1 20372.129,E2 20372.129} C_VEL
LIN {X 0,Y 417.371,Z 117.479,A -85,B 0,C 180,E1 20368.315,E2 20368.315} C_VEL
LIN {X 0,Y 417.359,Z 117.48,A -85,B 0,C 180,E1 20364.448,E2 20364.448} C_VEL
LIN {X 0,Y 417.338,Z 117.499,A -85,B 0,C 180,E1 20360.767,E2 20360.767} C_VEL
LIN {X 0,Y 417.328,Z 117.495,A -85,B 0,C 180,E1 20356.995,E2 20356.995} C_VEL
LIN {X 0,Y 417.317,Z 117.476,A -85,B 0,C 180,E1 20353.297,E2 20353.297} C_VEL
LIN {X 0,Y 417.318,Z 117.498,A -85,B 0,C 180,E1 20349.376,E2 20349.376} C_VEL
LIN {X 0,Y 417.318,Z 117.495,A -85,B 0,C 180,E1 20345.499,E2 20345.499} C_VEL
LIN {X 0,Y 417.318,Z 117.48,A -85,B 0,C 180,E1 20341.647,E2 20341.647} C_VEL
LIN {X 0,Y 417.331,Z 117.501,A -85,B 0,C 180,E1 20337.94,E2 20337.94} C_VEL
LIN {X 0,Y 417.346,Z 117.475,A -85,B 0,C 180,E1 20334.225,E2 20334.225} C_VEL
LIN {X 0,Y 417.359,Z 117.493,A -85,B 0,C 180,E1 20330.485,E2 20330.485} C_VEL
LIN {X 0,Y 417.362,Z 117.488,A -85,B 0,C 180,E1 20326.561,E2 20326.561} C_VEL
LIN {X 0,Y 417.349,Z 117.476,A -85,B 0,C 180,E1 20322.718,E2 20322.718} C_VEL
LIN {X 0,Y 417.338,Z 117.501,A -85,B 0,C 180,E1 20318.938,E2 20318.938} C_VEL
LIN {X 0,Y 417.32,Z 117.492,A -85,B 0,C 180,E1 20315.21,E2 20315.21} C_VEL
LIN {X 0,Y 417.309,Z 117.479,A -85,B 0,C 180,E1 20311.523,E2 20311.523} C_VEL
LIN {X 0,Y 417.308,Z 117.491,A -85,B 0,C 180,E1 20307.703,E2 20307.703} C_VEL
LIN {X 0,Y 417.309,Z 117.499,A -85,B 0,C 180,E1 20303.845,E2 20303.845} C_VEL
LIN {X 0,Y 417.313,Z 117.499,A -85,B 0,C 180,E1 20300.05,E2 20300.05} C_VEL
LIN {X 0,Y 417.328,Z 117.492,A -85,B 0,C 180,E1 20296.347,E2 20296.347} C_VEL
LIN {X 0,Y 417.337,Z 117.491,A -85,B 0,C 180,E1 20292.501,E2 20292.501} C_VEL
LIN {X 0,Y 417.327,Z 117.634,A -85,B 0,C 180,E1 20292.008,E2 20292.008} C_VEL
LIN {X 0,Y 418.603,Z 120.962,A -85,B 0,C 180,E1 20291.408,E2 20291.408} C_VEL
LIN {X 0,Y 424.753,Z 135.867,A -85,B 0,C 180,E1 20288.766,E2 20288.766} C_VEL
LIN {X 0,Y 430.896,Z 152.276,A -85,B 0,C 180,E1 20286.112,E2 20286.112} C_VEL
LIN {X 0,Y 435.077,Z 165.199,A -85,B 0,C 180,E1 20284.213,E2 20284.213} C_VEL
LIN {X 0,Y 434.338,Z 173.699,A -85,B 0,C 180,E1 20283.378,E2 20283.378} C_VEL
LIN {X 0,Y 439.832,Z 206.239,A -85,B 0,C 180,E1 20282.249,E2 20282.249} C_VEL
LIN {X 0,Y 436.496,Z 391.565,A -85,B 0,C 180,E1 20279.244,E2 20279.244} C_VEL
LIN {X 0,Y 435.599,Z 410.73,A -85,B 0,C 180,E1 20278.693,E2 20278.693} C_VEL
LIN {X 0,Y 434.954,Z 420.592,A -85,B 0,C 180,E1 20278.307,E2 20278.307} C_VEL
LIN {X 0,Y 433.509,Z 428.217,A -85,B 0,C 180,E1 20278.032,E2 20278.032} C_VEL
LIN {X 0,Y 426.929,Z 445.496,A -85,B 0,C 180,E1 20277.463,E2 20277.463} C_VEL
LIN {X 0,Y 425.099,Z 452.273,A -85,B 0,C 180,E1 20277.092,E2 20277.092} C_VEL
LIN {X 0,Y 424.972,Z 453.23,A -85,B 0,C 180,E1 20277.028,E2 20277.028} C_VEL
LIN {X 0,Y 422.891,Z 469.552,A -85,B 0,C 180,E1 20275.734,E2 20275.734} C_VEL
LIN {X 0,Y 420.727,Z 484.506,A -85,B 0,C 180,E1 20274.275,E2 20274.275} C_VEL
LIN {X 0,Y 418.434,Z 499,A -85,B 0,C 180,E1 20272.556,E2 20272.556} C_VEL
LIN {X 0,Y 416.243,Z 512.087,A -85,B 0,C 180,E1 20270.677,E2 20270.677} C_VEL
LIN {X 0,Y 414.18,Z 524.145,A -85,B 0,C 180,E1 20268.581,E2 20268.581} C_VEL
LIN {X 0,Y 412.389,Z 534.754,A -85,B 0,C 180,E1 20266.334,E2 20266.334} C_VEL
LIN {X 0,Y 410.879,Z 544.263,A -85,B 0,C 180,E1 20263.842,E2 20263.842} C_VEL
LIN {X 0,Y 409.754,Z 552.041,A -85,B 0,C 180,E1 20261.256,E2 20261.256} C_VEL
LIN {X 0,Y 409.007,Z 558.157,A -85,B 0,C 180,E1 20258.575,E2 20258.575} C_VEL
LIN {X 0,Y 408.57,Z 562.48,A -85,B 0,C 180,E1 20255.899,E2 20255.899} C_VEL
LIN {X 0,Y 408.353,Z 565.151,A -85,B 0,C 180,E1 20253.227,E2 20253.227} C_VEL
LIN {X 0,Y 408.286,Z 566.259,A -85,B 0,C 180,E1 20250.56,E2 20250.56} C_VEL
LIN {X 0,Y 408.316,Z 565.783,A -85,B 0,C 180,E1 20247.754,E2 20247.754} C_VEL
LIN {X 0,Y 408.475,Z 563.6,A -85,B 0,C 180,E1 20244.944,E2 20244.944} C_VEL
LIN {X 0,Y 408.823,Z 559.863,A -85,B 0,C 180,E1 20242.269,E2 20242.269} C_VEL
LIN {X 0,Y 409.451,Z 554.395,A -85,B 0,C 180,E1 20239.588,E2 20239.588} C_VEL
LIN {X 0,Y 410.406,Z 547.428,A -85,B 0,C 180,E1 20237.037,E2 20237.037} C_VEL
LIN {X 0,Y 411.71,Z 538.988,A -85,B 0,C 180,E1 20234.61,E2 20234.61} C_VEL
LIN {X 0,Y 413.395,Z 528.813,A -85,B 0,C 180,E1 20232.256,E2 20232.256} C_VEL
LIN {X 0,Y 415.299,Z 517.713,A -85,B 0,C 180,E1 20230.155,E2 20230.155} C_VEL
LIN {X 0,Y 417.523,Z 504.58,A -85,B 0,C 180,E1 20228.105,E2 20228.105} C_VEL
LIN {X 0,Y 419.862,Z 490.228,A -85,B 0,C 180,E1 20226.267,E2 20226.267} C_VEL
LIN {X 0,Y 422.123,Z 475.192,A -85,B 0,C 180,E1 20224.688,E2 20224.688} C_VEL
LIN {X 0,Y 424.25,Z 459.26,A -85,B 0,C 180,E1 20223.322,E2 20223.322} C_VEL
LIN {X 0,Y 426.186,Z 442.454,A -85,B 0,C 180,E1 20222.168,E2 20222.168} C_VEL
LIN {X 0,Y 427.84,Z 424.432,A -85,B 0,C 180,E1 20221.209,E2 20221.209} C_VEL
LIN {X 0,Y 429.124,Z 405.219,A -85,B 0,C 180,E1 20220.465,E2 20220.465} C_VEL
LIN {X 0,Y 429.896,Z 385.758,A -85,B 0,C 180,E1 20219.977,E2 20219.977} C_VEL
LIN {X 0,Y 433.233,Z 205.836,A -85,B 0,C 180,E1 20217.023,E2 20217.023} C_VEL
LIN {X 0,Y 427.577,Z 172.933,A -85,B 0,C 180,E1 20215.818,E2 20215.818} C_VEL
LIN {X 0,Y 427.992,Z 167.565,A -85,B 0,C 180,E1 20215.247,E2 20215.247} C_VEL
LIN {X 0,Y 421.981,Z 150.011,A -85,B 0,C 180,E1 20212.539,E2 20212.539} C_VEL
LIN {X 0,Y 415.529,Z 133.145,A -85,B 0,C 180,E1 20209.663,E2 20209.663} C_VEL
LIN {X 0,Y 410.657,Z 121.823,A -85,B 0,C 180,E1 20207.54,E2 20207.54} C_VEL
LIN {X 0,Y 409.421,Z 118.476,A -85,B 0,C 180,E1 20206.858,E2 20206.858} C_VEL
LIN {X 0,Y 409.431,Z 118.473,A -85,B 0,C 180,E1 20202.949,E2 20202.949} C_VEL
LIN {X 0,Y 409.455,Z 118.59,A -85,B 0,C 180,E1 20199.497,E2 20199.497} C_VEL
LIN {X 0,Y 419.157,Z 144.74,A -85,B 0,C 180,E1 20196.151,E2 20196.151} C_VEL
LIN {X 0,Y 424.705,Z 161.553,A -85,B 0,C 180,E1 20194.118,E2 20194.118} C_VEL
LIN {X 0,Y 423.701,Z 185.141,A -85,B 0,C 180,E1 20192.06,E2 20192.06} C_VEL
LIN {X 0,Y 426.31,Z 204.752,A -85,B 0,C 180,E1 20191.412,E2 20191.412} C_VEL
LIN {X 0,Y 420.589,Z 396.401,A -85,B 0,C 180,E1 20187.458,E2 20187.458} C_VEL
LIN {X 0,Y 419.783,Z 416.104,A -85,B 0,C 180,E1 20186.784,E2 20186.784} C_VEL
LIN {X 0,Y 418.768,Z 434.41,A -85,B 0,C 180,E1 20185.909,E2 20185.909} C_VEL
LIN {X 0,Y 417.514,Z 452.579,A -85,B 0,C 180,E1 20184.777,E2 20184.777} C_VEL
LIN {X 0,Y 416.086,Z 470.588,A -85,B 0,C 180,E1 20183.36,E2 20183.36} C_VEL
LIN {X 0,Y 414.676,Z 486.672,A -85,B 0,C 180,E1 20181.797,E2 20181.797} C_VEL
LIN {X 0,Y 413.278,Z 501.742,A -85,B 0,C 180,E1 20180.02,E2 20180.02} C_VEL
